/POS
P[2158]{
   GP1:
	UF : 7, UT : 3,	CONFIG : 'F U T, 0, 0, 0',
	X =   169.241  mm,	Y =   268.585  mm,	Z =     0.000  mm,
	W =  -167.363 deg,	P =     0.002 deg,	R =   163.143 deg
};
P[2159]{
   GP1:
	UF : 7, UT : 3,	CONFIG : 'F U T, 0, 0, 0',
	X =   183.720  mm,	Y =   258.920  mm,	Z =     0.001  mm,
	W =  -167.363 deg,	P =     0.001 deg,	R =   159.718 deg
};
P[2160]{
   GP1:
	UF : 7, UT : 3,	CONFIG : 'F U T, 0, 0, 0',
	X =   198.126  mm,	Y =   248.045  mm,	Z =     0.001  mm,
	W =  -167.364 deg,	P =     0.000 deg,	R =   156.405 deg
};
P[2161]{
   GP1:
	UF : 7, UT : 3,	CONFIG : 'F U T, 0, 0, 0',
	X =   212.090  mm,	Y =   236.233  mm,	Z =     0.001  mm,
	W =  -167.364 deg,	P =    -0.002 deg,	R =   153.153 deg
};
P[2162]{
   GP1:
	UF : 7, UT : 3,	CONFIG : 'F U T, 0, 0, 0',
	X =   224.191  mm,	Y =   224.763  mm,	Z =     0.000  mm,
	W =  -167.364 deg,	P =    -0.003 deg,	R =   149.479 deg
};
P[2163]{
   GP1:
	UF : 7, UT : 3,	CONFIG : 'F U T, 0, 0, 0',
	X =   224.191  mm,	Y =   224.763  mm,	Z =     0.000  mm,
	W =  -167.364 deg,	P =    -0.003 deg,	R =   149.479 deg
};
P[2164]{
   GP1:
	UF : 7, UT : 3,	CONFIG : 'F U T, 0, 0, 0',
	X =   224.191  mm,	Y =   224.763  mm,	Z =     0.000  mm,
	W =  -167.364 deg,	P =    -0.003 deg,	R =   149.479 deg
};
P[2165]{
   GP1:
	UF : 7, UT : 3,	CONFIG : 'F U T, 0, 0, 0',
	X =   224.191  mm,	Y =   224.763  mm,	Z =     0.000  mm,
	W =  -167.364 deg,	P =    -0.003 deg,	R =   149.479 deg
};
P[2166]{
   GP1:
	UF : 7, UT : 3,	CONFIG : 'F U T, 0, 0, 0',
	X =   269.018  mm,	Y =   168.557  mm,	Z =     0.000  mm,
	W =  -167.363 deg,	P =     0.003 deg,	R =   137.473 deg
};
P[2167]{
   GP1:
	UF : 7, UT : 3,	CONFIG : 'F U T, 0, 0, 0',
	X =   269.018  mm,	Y =   168.557  mm,	Z =     0.000  mm,
	W =  -167.363 deg,	P =     0.003 deg,	R =   137.473 deg
};
P[2168]{
   GP1:
	UF : 7, UT : 3,	CONFIG : 'F U T, 0, 0, 0',
	X =   269.018  mm,	Y =   168.557  mm,	Z =     0.000  mm,
	W =  -167.363 deg,	P =     0.003 deg,	R =   137.473 deg
};
P[2169]{
   GP1:
	UF : 7, UT : 3,	CONFIG : 'F U T, 0, 0, 0',
	X =   269.018  mm,	Y =   168.557  mm,	Z =     0.000  mm,
	W =  -167.363 deg,	P =     0.003 deg,	R =   137.473 deg
};
P[2170]{
   GP1:
	UF : 7, UT : 3,	CONFIG : 'F U T, 0, 0, 0',
	X =   277.589  mm,	Y =   154.047  mm,	Z =     0.001  mm,
	W =  -167.363 deg,	P =     0.001 deg,	R =   134.070 deg
};
P[2171]{
   GP1:
	UF : 7, UT : 3,	CONFIG : 'F U T, 0, 0, 0',
	X =   285.805  mm,	Y =   138.195  mm,	Z =     0.001  mm,
	W =  -167.364 deg,	P =     0.000 deg,	R =   130.902 deg
};
P[2172]{
   GP1:
	UF : 7, UT : 3,	CONFIG : 'F U T, 0, 0, 0',
	X =   292.963  mm,	Y =   122.300  mm,	Z =     0.001  mm,
	W =  -167.364 deg,	P =    -0.001 deg,	R =   127.666 deg
};
P[2173]{
   GP1:
	UF : 7, UT : 3,	CONFIG : 'F U T, 0, 0, 0',
	X =   299.514  mm,	Y =   105.233  mm,	Z =     0.000  mm,
	W =  -167.364 deg,	P =    -0.003 deg,	R =   124.545 deg
};
P[2174]{
   GP1:
	UF : 7, UT : 3,	CONFIG : 'F U T, 0, 0, 0',
	X =   299.514  mm,	Y =   105.233  mm,	Z =     0.000  mm,
	W =  -167.364 deg,	P =    -0.003 deg,	R =   124.545 deg
};
P[2175]{
   GP1:
	UF : 7, UT : 3,	CONFIG : 'F U T, 0, 0, 0',
	X =   299.514  mm,	Y =   105.233  mm,	Z =     0.000  mm,
	W =  -167.364 deg,	P =    -0.003 deg,	R =   124.545 deg
};
P[2176]{
   GP1:
	UF : 7, UT : 3,	CONFIG : 'F U T, 0, 0, 0',
	X =   299.514  mm,	Y =   105.233  mm,	Z =     0.000  mm,
	W =  -167.364 deg,	P =    -0.003 deg,	R =   124.545 deg
};
P[2177]{
   GP1:
	UF : 7, UT : 3,	CONFIG : 'F U T, 0, 0, 0',
	X =   315.526  mm,	Y =    35.143  mm,	Z =     0.000  mm,
	W =  -167.363 deg,	P =     0.001 deg,	R =   110.775 deg
};
P[2178]{
   GP1:
	UF : 7, UT : 3,	CONFIG : 'F U T, 0, 0, 0',
	X =   315.526  mm,	Y =    35.143  mm,	Z =     0.000  mm,
	W =  -167.363 deg,	P =     0.001 deg,	R =   110.775 deg
};
P[2179]{
   GP1:
	UF : 7, UT : 3,	CONFIG : 'F U T, 0, 0, 0',
	X =   315.526  mm,	Y =    35.143  mm,	Z =     0.000  mm,
	W =  -167.363 deg,	P =     0.001 deg,	R =   110.775 deg
};
P[2180]{
   GP1:
	UF : 7, UT : 3,	CONFIG : 'F U T, 0, 0, 0',
	X =   315.526  mm,	Y =    35.143  mm,	Z =     0.000  mm,
	W =  -167.363 deg,	P =     0.001 deg,	R =   110.775 deg
};
P[2181]{
   GP1:
	UF : 7, UT : 3,	CONFIG : 'F U T, 0, 0, 0',
	X =   316.958  mm,	Y =    17.828  mm,	Z =     0.000  mm,
	W =  -167.363 deg,	P =     0.000 deg,	R =   108.286 deg
};
P[2182]{
   GP1:
	UF : 7, UT : 3,	CONFIG : 'F U T, 0, 0, 0',
	X =   317.478  mm,	Y =     0.000  mm,	Z =     0.000  mm,
	W =  -167.364 deg,	P =    -0.001 deg,	R =   105.693 deg
};
P[2183]{
   GP1:
	UF : 7, UT : 3,	CONFIG : 'F U T, 0, 0, 0',
	X =   317.478  mm,	Y =     0.000  mm,	Z =     0.000  mm,
	W =  -167.364 deg,	P =    -0.001 deg,	R =   105.693 deg
};
P[2184]{
   GP1:
	UF : 7, UT : 3,	CONFIG : 'F U T, 0, 0, 0',
	X =   317.478  mm,	Y =     0.000  mm,	Z =     0.000  mm,
	W =  -167.364 deg,	P =    -0.001 deg,	R =   105.693 deg
};
P[2185]{
   GP1:
	UF : 7, UT : 3,	CONFIG : 'F U T, 0, 0, 0',
	X =   317.478  mm,	Y =     0.000  mm,	Z =     0.000  mm,
	W =  -167.364 deg,	P =    -0.001 deg,	R =   105.693 deg
};
P[2186]{
   GP1:
	UF : 7, UT : 3,	CONFIG : 'F U T, 0, 0, 0',
	X =   314.344  mm,	Y =     0.000  mm,	Z =     0.000  mm,
	W =  -167.364 deg,	P =    -0.001 deg,	R =   105.705 deg
};
P[2187]{
   GP1:
	UF : 7, UT : 3,	CONFIG : 'F U T, 0, 0, 0',
	X =   314.344  mm,	Y =     0.000  mm,	Z =     0.000  mm,
	W =  -167.364 deg,	P =    -0.001 deg,	R =   105.705 deg
};
P[2188]{
   GP1:
	UF : 7, UT : 3,	CONFIG : 'F U T, 0, 0, 0',
	X =   314.344  mm,	Y =     0.000  mm,	Z =     0.000  mm,
	W =  -167.364 deg,	P =    -0.001 deg,	R =   105.705 deg
};
P[2189]{
   GP1:
	UF : 7, UT : 3,	CONFIG : 'F U T, 0, 0, 0',
	X =   314.344  mm,	Y =     0.000  mm,	Z =     0.000  mm,
	W =  -167.364 deg,	P =    -0.001 deg,	R =   105.705 deg
};
P[2190]{
   GP1:
	UF : 7, UT : 3,	CONFIG : 'F U T, 0, 0, 0',
	X =   313.796  mm,	Y =    18.258  mm,	Z =     0.000  mm,
	W =  -167.363 deg,	P =     0.000 deg,	R =   108.359 deg
};
P[2191]{
   GP1:
	UF : 7, UT : 3,	CONFIG : 'F U T, 0, 0, 0',
	X =   312.363  mm,	Y =    35.193  mm,	Z =     0.000  mm,
	W =  -167.363 deg,	P =     0.001 deg,	R =   111.081 deg
};
P[2192]{
   GP1:
	UF : 7, UT : 3,	CONFIG : 'F U T, 0, 0, 0',
	X =   312.363  mm,	Y =    35.193  mm,	Z =     0.000  mm,
	W =  -167.363 deg,	P =     0.001 deg,	R =   111.081 deg
};
P[2193]{
   GP1:
	UF : 7, UT : 3,	CONFIG : 'F U T, 0, 0, 0',
	X =   312.363  mm,	Y =    35.193  mm,	Z =     0.000  mm,
	W =  -167.363 deg,	P =     0.001 deg,	R =   111.081 deg
};
P[2194]{
   GP1:
	UF : 7, UT : 3,	CONFIG : 'F U T, 0, 0, 0',
	X =   312.363  mm,	Y =    35.193  mm,	Z =     0.000  mm,
	W =  -167.363 deg,	P =     0.001 deg,	R =   111.081 deg
};
P[2195]{
   GP1:
	UF : 7, UT : 3,	CONFIG : 'F U T, 0, 0, 0',
	X =   296.692  mm,	Y =   103.818  mm,	Z =     0.000  mm,
	W =  -167.364 deg,	P =    -0.003 deg,	R =   124.612 deg
};
P[2196]{
   GP1:
	UF : 7, UT : 3,	CONFIG : 'F U T, 0, 0, 0',
	X =   296.692  mm,	Y =   103.818  mm,	Z =     0.000  mm,
	W =  -167.364 deg,	P =    -0.003 deg,	R =   124.612 deg
};
P[2197]{
   GP1:
	UF : 7, UT : 3,	CONFIG : 'F U T, 0, 0, 0',
	X =   296.692  mm,	Y =   103.818  mm,	Z =     0.000  mm,
	W =  -167.364 deg,	P =    -0.003 deg,	R =   124.612 deg
};
P[2198]{
   GP1:
	UF : 7, UT : 3,	CONFIG : 'F U T, 0, 0, 0',
	X =   296.692  mm,	Y =   103.818  mm,	Z =     0.000  mm,
	W =  -167.364 deg,	P =    -0.003 deg,	R =   124.612 deg
};
P[2199]{
   GP1:
	UF : 7, UT : 3,	CONFIG : 'F U T, 0, 0, 0',
	X =   289.976  mm,	Y =   121.319  mm,	Z =     0.001  mm,
	W =  -167.364 deg,	P =    -0.001 deg,	R =   127.739 deg
};
P[2200]{
   GP1:
	UF : 7, UT : 3,	CONFIG : 'F U T, 0, 0, 0',
	X =   282.724  mm,	Y =   137.365  mm,	Z =     0.001  mm,
	W =  -167.363 deg,	P =     0.000 deg,	R =   130.985 deg
};
P[2201]{
   GP1:
	UF : 7, UT : 3,	CONFIG : 'F U T, 0, 0, 0',
	X =   274.534  mm,	Y =   153.088  mm,	Z =     0.001  mm,
	W =  -167.363 deg,	P =     0.001 deg,	R =   134.198 deg
};
P[2202]{
   GP1:
	UF : 7, UT : 3,	CONFIG : 'F U T, 0, 0, 0',
	X =   266.148  mm,	Y =   167.232  mm,	Z =     0.000  mm,
	W =  -167.362 deg,	P =     0.003 deg,	R =   137.749 deg
};
P[2203]{
   GP1:
	UF : 7, UT : 3,	CONFIG : 'F U T, 0, 0, 0',
	X =   266.148  mm,	Y =   167.232  mm,	Z =     0.000  mm,
	W =  -167.362 deg,	P =     0.003 deg,	R =   137.749 deg
};
P[2204]{
   GP1:
	UF : 7, UT : 3,	CONFIG : 'F U T, 0, 0, 0',
	X =   266.148  mm,	Y =   167.232  mm,	Z =     0.000  mm,
	W =  -167.362 deg,	P =     0.003 deg,	R =   137.749 deg
};
P[2205]{
   GP1:
	UF : 7, UT : 3,	CONFIG : 'F U T, 0, 0, 0',
	X =   266.148  mm,	Y =   167.232  mm,	Z =     0.000  mm,
	W =  -167.362 deg,	P =     0.003 deg,	R =   137.749 deg
};
P[2206]{
   GP1:
	UF : 7, UT : 3,	CONFIG : 'F U T, 0, 0, 0',
	X =   222.261  mm,	Y =   222.261  mm,	Z =     0.000  mm,
	W =  -167.364 deg,	P =    -0.003 deg,	R =   149.599 deg
};
P[2207]{
   GP1:
	UF : 7, UT : 3,	CONFIG : 'F U T, 0, 0, 0',
	X =   222.261  mm,	Y =   222.261  mm,	Z =     0.000  mm,
	W =  -167.364 deg,	P =    -0.003 deg,	R =   149.599 deg
};
P[2208]{
   GP1:
	UF : 7, UT : 3,	CONFIG : 'F U T, 0, 0, 0',
	X =   222.261  mm,	Y =   222.261  mm,	Z =     0.000  mm,
	W =  -167.364 deg,	P =    -0.003 deg,	R =   149.599 deg
};
P[2209]{
   GP1:
	UF : 7, UT : 3,	CONFIG : 'F U T, 0, 0, 0',
	X =   222.261  mm,	Y =   222.261  mm,	Z =     0.000  mm,
	W =  -167.364 deg,	P =    -0.003 deg,	R =   149.599 deg
};
P[2210]{
   GP1:
	UF : 7, UT : 3,	CONFIG : 'F U T, 0, 0, 0',
	X =   209.897  mm,	Y =   233.994  mm,	Z =     0.001  mm,
	W =  -167.364 deg,	P =    -0.002 deg,	R =   153.153 deg
};
P[2211]{
   GP1:
	UF : 7, UT : 3,	CONFIG : 'F U T, 0, 0, 0',
	X =   195.899  mm,	Y =   245.814  mm,	Z =     0.001  mm,
	W =  -167.363 deg,	P =     0.000 deg,	R =   156.411 deg
};
P[2212]{
   GP1:
	UF : 7, UT : 3,	CONFIG : 'F U T, 0, 0, 0',
	X =   181.688  mm,	Y =   256.510  mm,	Z =     0.001  mm,
	W =  -167.363 deg,	P =     0.001 deg,	R =   159.771 deg
};
P[2213]{
   GP1:
	UF : 7, UT : 3,	CONFIG : 'F U T, 0, 0, 0',
	X =   167.232  mm,	Y =   266.148  mm,	Z =     0.000  mm,
	W =  -167.362 deg,	P =     0.002 deg,	R =   163.242 deg
};
P[2214]{
   GP1:
	UF : 7, UT : 3,	CONFIG : 'F U T, 0, 0, 0',
	X =   167.232  mm,	Y =   266.148  mm,	Z =     0.000  mm,
	W =  -167.362 deg,	P =     0.002 deg,	R =   163.242 deg
};
P[2215]{
   GP1:
	UF : 7, UT : 3,	CONFIG : 'F U T, 0, 0, 0',
	X =   167.232  mm,	Y =   266.148  mm,	Z =     0.000  mm,
	W =  -167.362 deg,	P =     0.002 deg,	R =   163.242 deg
};
P[2216]{
   GP1:
	UF : 7, UT : 3,	CONFIG : 'F U T, 0, 0, 0',
	X =   167.232  mm,	Y =   266.148  mm,	Z =     0.000  mm,
	W =  -167.362 deg,	P =     0.002 deg,	R =   163.242 deg
};
P[2217]{
   GP1:
	UF : 7, UT : 3,	CONFIG : 'F U T, 0, 0, 0',
	X =   103.816  mm,	Y =   296.692  mm,	Z =     0.000  mm,
	W =  -167.364 deg,	P =    -0.001 deg,	R =   175.609 deg
};
P[2218]{
   GP1:
	UF : 7, UT : 3,	CONFIG : 'F U T, 0, 0, 0',
	X =   103.816  mm,	Y =   296.692  mm,	Z =     0.000  mm,
	W =  -167.364 deg,	P =    -0.001 deg,	R =   175.609 deg
};
P[2219]{
   GP1:
	UF : 7, UT : 3,	CONFIG : 'F U T, 0, 0, 0',
	X =   103.816  mm,	Y =   296.692  mm,	Z =     0.000  mm,
	W =  -167.364 deg,	P =    -0.001 deg,	R =   175.609 deg
};
P[2220]{
   GP1:
	UF : 7, UT : 3,	CONFIG : 'F U T, 0, 0, 0',
	X =   103.816  mm,	Y =   296.692  mm,	Z =     0.000  mm,
	W =  -167.364 deg,	P =    -0.001 deg,	R =   175.609 deg
};
P[2221]{
   GP1:
	UF : 7, UT : 3,	CONFIG : 'F U T, 0, 0, 0',
	X =    87.953  mm,	Y =   301.775  mm,	Z =     0.000  mm,
	W =  -167.364 deg,	P =    -0.001 deg,	R =   178.852 deg
};
P[2222]{
   GP1:
	UF : 7, UT : 3,	CONFIG : 'F U T, 0, 0, 0',
	X =    71.164  mm,	Y =   306.169  mm,	Z =     0.000  mm,
	W =  -167.363 deg,	P =     0.000 deg,	R =  -178.042 deg
};
P[2223]{
   GP1:
	UF : 7, UT : 3,	CONFIG : 'F U T, 0, 0, 0',
	X =    54.389  mm,	Y =   309.594  mm,	Z =     0.000  mm,
	W =  -167.363 deg,	P =     0.000 deg,	R =  -174.890 deg
};
P[2224]{
   GP1:
	UF : 7, UT : 3,	CONFIG : 'F U T, 0, 0, 0',
	X =    35.197  mm,	Y =   312.362  mm,	Z =     0.000  mm,
	W =  -167.363 deg,	P =     0.001 deg,	R =  -171.894 deg
};
P[2225]{
   GP1:
	UF : 7, UT : 3,	CONFIG : 'F U T, 0, 0, 0',
	X =    35.197  mm,	Y =   312.362  mm,	Z =     0.000  mm,
	W =  -167.363 deg,	P =     0.001 deg,	R =  -171.894 deg
};
P[2226]{
   GP1:
	UF : 7, UT : 3,	CONFIG : 'F U T, 0, 0, 0',
	X =    35.197  mm,	Y =   312.362  mm,	Z =     0.000  mm,
	W =  -167.363 deg,	P =     0.001 deg,	R =  -171.894 deg
};
P[2227]{
   GP1:
	UF : 7, UT : 3,	CONFIG : 'F U T, 0, 0, 0',
	X =    35.197  mm,	Y =   312.362  mm,	Z =     0.000  mm,
	W =  -167.363 deg,	P =     0.001 deg,	R =  -171.894 deg
};
P[2228]{
   GP1:
	UF : 7, UT : 3,	CONFIG : 'F U T, 0, 0, 0',
	X =   -35.197  mm,	Y =   312.362  mm,	Z =     0.000  mm,
	W =  -167.364 deg,	P =    -0.001 deg,	R =  -157.993 deg
};
P[2229]{
   GP1:
	UF : 7, UT : 3,	CONFIG : 'F U T, 0, 0, 0',
	X =   -35.197  mm,	Y =   312.362  mm,	Z =     0.000  mm,
	W =  -167.364 deg,	P =    -0.001 deg,	R =  -157.993 deg
};
P[2230]{
   GP1:
	UF : 7, UT : 3,	CONFIG : 'F U T, 0, 0, 0',
	X =   -35.197  mm,	Y =   312.362  mm,	Z =     0.000  mm,
	W =  -167.364 deg,	P =    -0.001 deg,	R =  -157.993 deg
};
P[2231]{
   GP1:
	UF : 7, UT : 3,	CONFIG : 'F U T, 0, 0, 0',
	X =   -35.197  mm,	Y =   312.362  mm,	Z =     0.000  mm,
	W =  -167.364 deg,	P =    -0.001 deg,	R =  -157.993 deg
};
P[2232]{
   GP1:
	UF : 7, UT : 3,	CONFIG : 'F U T, 0, 0, 0',
	X =   -54.397  mm,	Y =   309.592  mm,	Z =     0.001  mm,
	W =  -167.363 deg,	P =     0.000 deg,	R =  -154.999 deg
};
P[2233]{
   GP1:
	UF : 7, UT : 3,	CONFIG : 'F U T, 0, 0, 0',
	X =   -71.123  mm,	Y =   306.179  mm,	Z =     0.001  mm,
	W =  -167.363 deg,	P =     0.002 deg,	R =  -151.872 deg
};
P[2234]{
   GP1:
	UF : 7, UT : 3,	CONFIG : 'F U T, 0, 0, 0',
	X =   -87.830  mm,	Y =   301.810  mm,	Z =     0.001  mm,
	W =  -167.362 deg,	P =     0.003 deg,	R =  -148.771 deg
};
P[2235]{
   GP1:
	UF : 7, UT : 3,	CONFIG : 'F U T, 0, 0, 0',
	X =  -103.816  mm,	Y =   296.692  mm,	Z =     0.000  mm,
	W =  -167.361 deg,	P =     0.004 deg,	R =  -145.598 deg
};
P[2236]{
   GP1:
	UF : 7, UT : 3,	CONFIG : 'F U T, 0, 0, 0',
	X =  -103.816  mm,	Y =   296.692  mm,	Z =     0.000  mm,
	W =  -167.361 deg,	P =     0.004 deg,	R =  -145.598 deg
};
P[2237]{
   GP1:
	UF : 7, UT : 3,	CONFIG : 'F U T, 0, 0, 0',
	X =  -103.816  mm,	Y =   296.692  mm,	Z =     0.000  mm,
	W =  -167.361 deg,	P =     0.004 deg,	R =  -145.598 deg
};
P[2238]{
   GP1:
	UF : 7, UT : 3,	CONFIG : 'F U T, 0, 0, 0',
	X =  -103.816  mm,	Y =   296.692  mm,	Z =     0.000  mm,
	W =  -167.361 deg,	P =     0.004 deg,	R =  -145.598 deg
};
P[2239]{
   GP1:
	UF : 7, UT : 3,	CONFIG : 'F U T, 0, 0, 0',
	X =  -167.232  mm,	Y =   266.148  mm,	Z =     0.000  mm,
	W =  -167.365 deg,	P =    -0.022 deg,	R =  -132.938 deg
};
P[2240]{
   GP1:
	UF : 7, UT : 3,	CONFIG : 'F U T, 0, 0, 0',
	X =  -167.232  mm,	Y =   266.148  mm,	Z =     0.000  mm,
	W =  -167.365 deg,	P =    -0.022 deg,	R =  -132.938 deg
};
P[2241]{
   GP1:
	UF : 7, UT : 3,	CONFIG : 'F U T, 0, 0, 0',
	X =  -167.232  mm,	Y =   266.148  mm,	Z =     0.000  mm,
	W =  -167.365 deg,	P =    -0.022 deg,	R =  -132.938 deg
};
P[2242]{
   GP1:
	UF : 7, UT : 3,	CONFIG : 'F U T, 0, 0, 0',
	X =  -167.232  mm,	Y =   266.148  mm,	Z =     0.000  mm,
	W =  -167.365 deg,	P =    -0.022 deg,	R =  -132.938 deg
};
P[2243]{
   GP1:
	UF : 7, UT : 3,	CONFIG : 'F U T, 0, 0, 0',
	X =  -183.114  mm,	Y =   255.488  mm,	Z =     0.011  mm,
	W =  -167.354 deg,	P =    -0.024 deg,	R =  -129.291 deg
};
P[2244]{
   GP1:
	UF : 7, UT : 3,	CONFIG : 'F U T, 0, 0, 0',
	X =  -198.763  mm,	Y =   243.515  mm,	Z =     0.023  mm,
	W =  -167.343 deg,	P =    -0.029 deg,	R =  -125.737 deg
};
P[2245]{
   GP1:
	UF : 7, UT : 3,	CONFIG : 'F U T, 0, 0, 0',
	X =  -211.069  mm,	Y =   232.923  mm,	Z =     0.022  mm,
	W =  -167.329 deg,	P =     0.048 deg,	R =  -122.698 deg
};
P[2246]{
   GP1:
	UF : 7, UT : 3,	CONFIG : 'F U T, 0, 0, 0',
	X =  -222.261  mm,	Y =   222.261  mm,	Z =     0.000  mm,
	W =  -167.307 deg,	P =     0.119 deg,	R =  -119.437 deg
};
P[2247]{
   GP1:
	UF : 7, UT : 3,	CONFIG : 'F U T, 0, 0, 0',
	X =  -222.261  mm,	Y =   222.261  mm,	Z =     0.000  mm,
	W =  -167.307 deg,	P =     0.119 deg,	R =  -119.437 deg
};
P[2248]{
   GP1:
	UF : 7, UT : 3,	CONFIG : 'F U T, 0, 0, 0',
	X =  -222.261  mm,	Y =   222.261  mm,	Z =     0.000  mm,
	W =  -167.307 deg,	P =     0.119 deg,	R =  -119.437 deg
};
P[2249]{
   GP1:
	UF : 7, UT : 3,	CONFIG : 'F U T, 0, 0, 0',
	X =  -222.261  mm,	Y =   222.261  mm,	Z =     0.000  mm,
	W =  -167.307 deg,	P =     0.119 deg,	R =  -119.437 deg
};
P[2250]{
   GP1:
	UF : 7, UT : 3,	CONFIG : 'F U T, 0, 0, 0',
	X =  -266.148  mm,	Y =   167.232  mm,	Z =     0.000  mm,
	W =  -167.451 deg,	P =    -1.057 deg,	R =  -107.603 deg
};
P[2251]{
   GP1:
	UF : 7, UT : 3,	CONFIG : 'F U T, 0, 0, 0',
	X =  -266.148  mm,	Y =   167.232  mm,	Z =     0.000  mm,
	W =  -167.451 deg,	P =    -1.057 deg,	R =  -107.603 deg
};
P[2252]{
   GP1:
	UF : 7, UT : 3,	CONFIG : 'F U T, 0, 0, 0',
	X =  -266.148  mm,	Y =   167.232  mm,	Z =     0.000  mm,
	W =  -167.451 deg,	P =    -1.057 deg,	R =  -107.603 deg
};
P[2253]{
   GP1:
	UF : 7, UT : 3,	CONFIG : 'F U T, 0, 0, 0',
	X =  -266.148  mm,	Y =   167.232  mm,	Z =     0.000  mm,
	W =  -167.451 deg,	P =    -1.057 deg,	R =  -107.603 deg
};
P[2254]{
   GP1:
	UF : 7, UT : 3,	CONFIG : 'F U T, 0, 0, 0',
	X =  -269.323  mm,	Y =   162.065  mm,	Z =     0.117  mm,
	W =  -167.681 deg,	P =    -1.097 deg,	R =  -105.987 deg
};
P[2255]{
   GP1:
	UF : 7, UT : 3,	CONFIG : 'F U T, 0, 0, 0',
	X =  -277.022  mm,	Y =   148.536  mm,	Z =     0.388  mm,
	W =  -168.155 deg,	P =    -0.523 deg,	R =  -103.206 deg
};
P[2256]{
   GP1:
	UF : 7, UT : 3,	CONFIG : 'F U T, 0, 0, 0',
	X =  -285.722  mm,	Y =   131.011  mm,	Z =     0.439  mm,
	W =  -168.148 deg,	P =     0.621 deg,	R =   -99.624 deg
};
P[2257]{
   GP1:
	UF : 7, UT : 3,	CONFIG : 'F U T, 0, 0, 0',
	X =  -290.703  mm,	Y =   119.560  mm,	Z =     0.270  mm,
	W =  -167.700 deg,	P =     1.177 deg,	R =   -97.280 deg
};
P[2258]{
   GP1:
	UF : 7, UT : 3,	CONFIG : 'F U T, 0, 0, 0',
	X =  -292.713  mm,	Y =   114.575  mm,	Z =     0.169  mm,
	W =  -167.445 deg,	P =     1.139 deg,	R =   -96.303 deg
};
P[2259]{
   GP1:
	UF : 7, UT : 3,	CONFIG : 'F U T, 0, 0, 0',
	X =  -296.692  mm,	Y =   103.818  mm,	Z =     0.000  mm,
	W =  -167.160 deg,	P =     0.453 deg,	R =   -94.516 deg
};
P[2260]{
   GP1:
	UF : 7, UT : 3,	CONFIG : 'F U T, 0, 0, 0',
	X =  -296.692  mm,	Y =   103.818  mm,	Z =     0.000  mm,
	W =  -167.160 deg,	P =     0.453 deg,	R =   -94.516 deg
};
P[2261]{
   GP1:
	UF : 7, UT : 3,	CONFIG : 'F U T, 0, 0, 0',
	X =  -296.692  mm,	Y =   103.818  mm,	Z =     0.000  mm,
	W =  -167.160 deg,	P =     0.453 deg,	R =   -94.516 deg
};
P[2262]{
   GP1:
	UF : 7, UT : 3,	CONFIG : 'F U T, 0, 0, 0',
	X =  -296.692  mm,	Y =   103.818  mm,	Z =     0.000  mm,
	W =  -167.160 deg,	P =     0.453 deg,	R =   -94.516 deg
};
P[2263]{
   GP1:
	UF : 7, UT : 3,	CONFIG : 'F U T, 0, 1, 0',
	X =  -312.363  mm,	Y =    35.193  mm,	Z =     0.000  mm,
	W =  -167.364 deg,	P =    -0.010 deg,	R =   -80.974 deg
};
P[2264]{
   GP1:
	UF : 7, UT : 3,	CONFIG : 'F U T, 0, 1, 0',
	X =  -312.363  mm,	Y =    35.193  mm,	Z =     0.000  mm,
	W =  -167.364 deg,	P =    -0.010 deg,	R =   -80.974 deg
};
P[2265]{
   GP1:
	UF : 7, UT : 3,	CONFIG : 'F U T, 0, 1, 0',
	X =  -312.363  mm,	Y =    35.193  mm,	Z =     0.000  mm,
	W =  -167.364 deg,	P =    -0.010 deg,	R =   -80.974 deg
};
P[2266]{
   GP1:
	UF : 7, UT : 3,	CONFIG : 'F U T, 0, 1, 0',
	X =  -312.363  mm,	Y =    35.193  mm,	Z =     0.000  mm,
	W =  -167.364 deg,	P =    -0.010 deg,	R =   -80.974 deg
};
P[2267]{
   GP1:
	UF : 7, UT : 3,	CONFIG : 'F U T, 0, 1, 0',
	X =  -313.784  mm,	Y =    18.505  mm,	Z =     0.001  mm,
	W =  -167.364 deg,	P =    -0.002 deg,	R =   -78.279 deg
};
P[2268]{
   GP1:
	UF : 7, UT : 3,	CONFIG : 'F U T, 0, 1, 0',
	X =  -314.344  mm,	Y =     0.000  mm,	Z =     0.000  mm,
	W =  -167.362 deg,	P =     0.006 deg,	R =   -75.585 deg
};
P[2269]{
   GP1:
	UF : 7, UT : 3,	CONFIG : 'F U T, 0, 1, 0',
	X =  -314.344  mm,	Y =     0.000  mm,	Z =     0.000  mm,
	W =  -167.362 deg,	P =     0.006 deg,	R =   -75.585 deg
};
P[2270]{
   GP1:
	UF : 7, UT : 3,	CONFIG : 'F U T, 0, 1, 0',
	X =  -314.344  mm,	Y =     0.000  mm,	Z =     0.000  mm,
	W =  -167.362 deg,	P =     0.006 deg,	R =   -75.585 deg
};
P[2271]{
   GP1:
	UF : 7, UT : 3,	CONFIG : 'F U T, 0, 1, 0',
	X =  -314.344  mm,	Y =     0.000  mm,	Z =     0.000  mm,
	W =  -167.362 deg,	P =     0.006 deg,	R =   -75.585 deg
};
P[2272]{
   GP1:
	UF : 7, UT : 3,	CONFIG : 'F U T, 0, 1, 0',
	X =  -311.210  mm,	Y =     0.000  mm,	Z =     0.000  mm,
	W =  -167.362 deg,	P =     0.005 deg,	R =   -75.574 deg
};
P[2273]{
   GP1:
	UF : 7, UT : 3,	CONFIG : 'F U T, 0, 1, 0',
	X =  -311.210  mm,	Y =     0.000  mm,	Z =     0.000  mm,
	W =  -167.362 deg,	P =     0.005 deg,	R =   -75.574 deg
};
P[2274]{
   GP1:
	UF : 7, UT : 3,	CONFIG : 'F U T, 0, 1, 0',
	X =  -311.210  mm,	Y =     0.000  mm,	Z =     0.000  mm,
	W =  -167.362 deg,	P =     0.005 deg,	R =   -75.574 deg
};
P[2275]{
   GP1:
	UF : 7, UT : 3,	CONFIG : 'F U T, 0, 1, 0',
	X =  -311.210  mm,	Y =     0.000  mm,	Z =     0.000  mm,
	W =  -167.362 deg,	P =     0.005 deg,	R =   -75.574 deg
};
P[2276]{
   GP1:
	UF : 7, UT : 3,	CONFIG : 'F U T, 0, 1, 0',
	X =  -310.609  mm,	Y =    19.167  mm,	Z =     0.001  mm,
	W =  -167.363 deg,	P =    -0.003 deg,	R =   -78.435 deg
};
P[2277]{
   GP1:
	UF : 7, UT : 3,	CONFIG : 'F U T, 0, 1, 0',
	X =  -309.165  mm,	Y =    35.521  mm,	Z =     0.000  mm,
	W =  -167.364 deg,	P =    -0.010 deg,	R =   -81.404 deg
};
P[2278]{
   GP1:
	UF : 7, UT : 3,	CONFIG : 'F U T, 0, 1, 0',
	X =  -309.165  mm,	Y =    35.521  mm,	Z =     0.000  mm,
	W =  -167.364 deg,	P =    -0.010 deg,	R =   -81.404 deg
};
P[2279]{
   GP1:
	UF : 7, UT : 3,	CONFIG : 'F U T, 0, 1, 0',
	X =  -309.165  mm,	Y =    35.521  mm,	Z =     0.000  mm,
	W =  -167.364 deg,	P =    -0.010 deg,	R =   -81.404 deg
};
P[2280]{
   GP1:
	UF : 7, UT : 3,	CONFIG : 'F U T, 0, 1, 0',
	X =  -309.165  mm,	Y =    35.521  mm,	Z =     0.000  mm,
	W =  -167.364 deg,	P =    -0.010 deg,	R =   -81.404 deg
};
P[2281]{
   GP1:
	UF : 7, UT : 3,	CONFIG : 'F U T, 0, 0, 0',
	X =  -293.963  mm,	Y =   102.140  mm,	Z =     0.000  mm,
	W =  -167.168 deg,	P =     0.349 deg,	R =   -94.592 deg
};
P[2282]{
   GP1:
	UF : 7, UT : 3,	CONFIG : 'F U T, 0, 0, 0',
	X =  -293.963  mm,	Y =   102.140  mm,	Z =     0.000  mm,
	W =  -167.168 deg,	P =     0.349 deg,	R =   -94.592 deg
};
P[2283]{
   GP1:
	UF : 7, UT : 3,	CONFIG : 'F U T, 0, 0, 0',
	X =  -293.963  mm,	Y =   102.140  mm,	Z =     0.000  mm,
	W =  -167.168 deg,	P =     0.349 deg,	R =   -94.592 deg
};
P[2284]{
   GP1:
	UF : 7, UT : 3,	CONFIG : 'F U T, 0, 0, 0',
	X =  -293.963  mm,	Y =   102.140  mm,	Z =     0.000  mm,
	W =  -167.168 deg,	P =     0.349 deg,	R =   -94.592 deg
};
P[2285]{
   GP1:
	UF : 7, UT : 3,	CONFIG : 'F U T, 0, 0, 0',
	X =  -289.713  mm,	Y =   113.629  mm,	Z =     0.153  mm,
	W =  -167.448 deg,	P =     0.997 deg,	R =   -96.337 deg
};
P[2286]{
   GP1:
	UF : 7, UT : 3,	CONFIG : 'F U T, 0, 0, 0',
	X =  -285.444  mm,	Y =   123.944  mm,	Z =     0.328  mm,
	W =  -167.908 deg,	P =     0.905 deg,	R =   -98.395 deg
};
P[2287]{
   GP1:
	UF : 7, UT : 3,	CONFIG : 'F U T, 0, 0, 0',
	X =  -278.233  mm,	Y =   139.399  mm,	Z =     0.413  mm,
	W =  -168.175 deg,	P =     0.054 deg,	R =  -101.560 deg
};
P[2288]{
   GP1:
	UF : 7, UT : 3,	CONFIG : 'F U T, 0, 0, 0',
	X =  -270.057  mm,	Y =   154.632  mm,	Z =     0.235  mm,
	W =  -167.853 deg,	P =    -0.831 deg,	R =  -104.757 deg
};
P[2289]{
   GP1:
	UF : 7, UT : 3,	CONFIG : 'F U T, 0, 0, 0',
	X =  -263.128  mm,	Y =   166.143  mm,	Z =     0.000  mm,
	W =  -167.353 deg,	P =    -0.982 deg,	R =  -107.921 deg
};
P[2290]{
   GP1:
	UF : 7, UT : 3,	CONFIG : 'F U T, 0, 0, 0',
	X =  -263.128  mm,	Y =   166.143  mm,	Z =     0.000  mm,
	W =  -167.353 deg,	P =    -0.982 deg,	R =  -107.921 deg
};
P[2291]{
   GP1:
	UF : 7, UT : 3,	CONFIG : 'F U T, 0, 0, 0',
	X =  -263.128  mm,	Y =   166.143  mm,	Z =     0.000  mm,
	W =  -167.353 deg,	P =    -0.982 deg,	R =  -107.921 deg
};
P[2292]{
   GP1:
	UF : 7, UT : 3,	CONFIG : 'F U T, 0, 0, 0',
	X =  -263.128  mm,	Y =   166.143  mm,	Z =     0.000  mm,
	W =  -167.353 deg,	P =    -0.982 deg,	R =  -107.921 deg
};
P[2293]{
   GP1:
	UF : 7, UT : 3,	CONFIG : 'F U T, 0, 0, 0',
	X =  -220.529  mm,	Y =   219.561  mm,	Z =     0.000  mm,
	W =  -167.294 deg,	P =     0.118 deg,	R =  -119.493 deg
};
P[2294]{
   GP1:
	UF : 7, UT : 3,	CONFIG : 'F U T, 0, 0, 0',
	X =  -220.529  mm,	Y =   219.561  mm,	Z =     0.000  mm,
	W =  -167.294 deg,	P =     0.118 deg,	R =  -119.493 deg
};
P[2295]{
   GP1:
	UF : 7, UT : 3,	CONFIG : 'F U T, 0, 0, 0',
	X =  -220.529  mm,	Y =   219.561  mm,	Z =     0.000  mm,
	W =  -167.294 deg,	P =     0.118 deg,	R =  -119.493 deg
};
P[2296]{
   GP1:
	UF : 7, UT : 3,	CONFIG : 'F U T, 0, 0, 0',
	X =  -220.529  mm,	Y =   219.561  mm,	Z =     0.000  mm,
	W =  -167.294 deg,	P =     0.118 deg,	R =  -119.493 deg
};
P[2297]{
   GP1:
	UF : 7, UT : 3,	CONFIG : 'F U T, 0, 0, 0',
	X =  -208.972  mm,	Y =   230.595  mm,	Z =     0.023  mm,
	W =  -167.322 deg,	P =     0.047 deg,	R =  -122.742 deg
};
P[2298]{
   GP1:
	UF : 7, UT : 3,	CONFIG : 'F U T, 0, 0, 0',
	X =  -196.378  mm,	Y =   241.419  mm,	Z =     0.024  mm,
	W =  -167.342 deg,	P =    -0.031 deg,	R =  -125.847 deg
};
P[2299]{
   GP1:
	UF : 7, UT : 3,	CONFIG : 'F U T, 0, 0, 0',
	X =  -181.152  mm,	Y =   253.038  mm,	Z =     0.012  mm,
	W =  -167.352 deg,	P =    -0.027 deg,	R =  -129.328 deg
};
P[2300]{
   GP1:
	UF : 7, UT : 3,	CONFIG : 'F U T, 0, 0, 0',
	X =  -164.987  mm,	Y =   263.859  mm,	Z =     0.000  mm,
	W =  -167.364 deg,	P =    -0.024 deg,	R =  -132.775 deg
};
P[2301]{
   GP1:
	UF : 7, UT : 3,	CONFIG : 'F U T, 0, 0, 0',
	X =  -164.987  mm,	Y =   263.859  mm,	Z =     0.000  mm,
	W =  -167.364 deg,	P =    -0.024 deg,	R =  -132.775 deg
};
P[2302]{
   GP1:
	UF : 7, UT : 3,	CONFIG : 'F U T, 0, 0, 0',
	X =  -164.987  mm,	Y =   263.859  mm,	Z =     0.000  mm,
	W =  -167.364 deg,	P =    -0.024 deg,	R =  -132.775 deg
};
P[2303]{
   GP1:
	UF : 7, UT : 3,	CONFIG : 'F U T, 0, 0, 0',
	X =  -164.987  mm,	Y =   263.859  mm,	Z =     0.000  mm,
	W =  -167.364 deg,	P =    -0.024 deg,	R =  -132.775 deg
};
P[2304]{
   GP1:
	UF : 7, UT : 3,	CONFIG : 'F U T, 0, 0, 0',
	X =  -103.426  mm,	Y =   293.504  mm,	Z =     0.000  mm,
	W =  -167.361 deg,	P =     0.005 deg,	R =  -145.207 deg
};
P[2305]{
   GP1:
	UF : 7, UT : 3,	CONFIG : 'F U T, 0, 0, 0',
	X =  -103.426  mm,	Y =   293.504  mm,	Z =     0.000  mm,
	W =  -167.361 deg,	P =     0.005 deg,	R =  -145.207 deg
};
P[2306]{
   GP1:
	UF : 7, UT : 3,	CONFIG : 'F U T, 0, 0, 0',
	X =  -103.426  mm,	Y =   293.504  mm,	Z =     0.000  mm,
	W =  -167.361 deg,	P =     0.005 deg,	R =  -145.207 deg
};
P[2307]{
   GP1:
	UF : 7, UT : 3,	CONFIG : 'F U T, 0, 0, 0',
	X =  -103.426  mm,	Y =   293.504  mm,	Z =     0.000  mm,
	W =  -167.361 deg,	P =     0.005 deg,	R =  -145.207 deg
};
P[2308]{
   GP1:
	UF : 7, UT : 3,	CONFIG : 'F U T, 0, 0, 0',
	X =   -87.653  mm,	Y =   298.599  mm,	Z =     0.001  mm,
	W =  -167.362 deg,	P =     0.003 deg,	R =  -148.621 deg
};
P[2309]{
   GP1:
	UF : 7, UT : 3,	CONFIG : 'F U T, 0, 0, 0',
	X =   -70.707  mm,	Y =   303.056  mm,	Z =     0.001  mm,
	W =  -167.362 deg,	P =     0.002 deg,	R =  -151.841 deg
};
P[2310]{
   GP1:
	UF : 7, UT : 3,	CONFIG : 'F U T, 0, 0, 0',
	X =   -53.533  mm,	Y =   306.560  mm,	Z =     0.001  mm,
	W =  -167.363 deg,	P =     0.000 deg,	R =  -155.049 deg
};
P[2311]{
   GP1:
	UF : 7, UT : 3,	CONFIG : 'F U T, 0, 0, 0',
	X =   -34.169  mm,	Y =   309.326  mm,	Z =     0.000  mm,
	W =  -167.363 deg,	P =    -0.002 deg,	R =  -158.094 deg
};
P[2312]{
   GP1:
	UF : 7, UT : 3,	CONFIG : 'F U T, 0, 0, 0',
	X =   -34.169  mm,	Y =   309.326  mm,	Z =     0.000  mm,
	W =  -167.363 deg,	P =    -0.002 deg,	R =  -158.094 deg
};
P[2313]{
   GP1:
	UF : 7, UT : 3,	CONFIG : 'F U T, 0, 0, 0',
	X =   -34.169  mm,	Y =   309.326  mm,	Z =     0.000  mm,
	W =  -167.363 deg,	P =    -0.002 deg,	R =  -158.094 deg
};
P[2314]{
   GP1:
	UF : 7, UT : 3,	CONFIG : 'F U T, 0, 0, 0',
	X =   -34.169  mm,	Y =   309.326  mm,	Z =     0.000  mm,
	W =  -167.363 deg,	P =    -0.002 deg,	R =  -158.094 deg
};
P[2315]{
   GP1:
	UF : 7, UT : 3,	CONFIG : 'F U T, 0, 0, 0',
	X =    34.169  mm,	Y =   309.326  mm,	Z =     0.000  mm,
	W =  -167.363 deg,	P =     0.001 deg,	R =  -171.797 deg
};
P[2316]{
   GP1:
	UF : 7, UT : 3,	CONFIG : 'F U T, 0, 0, 0',
	X =    34.169  mm,	Y =   309.326  mm,	Z =     0.000  mm,
	W =  -167.363 deg,	P =     0.001 deg,	R =  -171.797 deg
};
P[2317]{
   GP1:
	UF : 7, UT : 3,	CONFIG : 'F U T, 0, 0, 0',
	X =    34.169  mm,	Y =   309.326  mm,	Z =     0.000  mm,
	W =  -167.363 deg,	P =     0.001 deg,	R =  -171.797 deg
};
P[2318]{
   GP1:
	UF : 7, UT : 3,	CONFIG : 'F U T, 0, 0, 0',
	X =    34.169  mm,	Y =   309.326  mm,	Z =     0.000  mm,
	W =  -167.363 deg,	P =     0.001 deg,	R =  -171.797 deg
};
P[2319]{
   GP1:
	UF : 7, UT : 3,	CONFIG : 'F U T, 0, 0, 0',
	X =    53.482  mm,	Y =   306.568  mm,	Z =     0.000  mm,
	W =  -167.363 deg,	P =     0.000 deg,	R =  -174.856 deg
};
P[2320]{
   GP1:
	UF : 7, UT : 3,	CONFIG : 'F U T, 0, 0, 0',
	X =    70.739  mm,	Y =   303.048  mm,	Z =     0.000  mm,
	W =  -167.363 deg,	P =     0.000 deg,	R =  -178.048 deg
};
P[2321]{
   GP1:
	UF : 7, UT : 3,	CONFIG : 'F U T, 0, 0, 0',
	X =    87.613  mm,	Y =   298.610  mm,	Z =     0.000  mm,
	W =  -167.363 deg,	P =    -0.001 deg,	R =   178.718 deg
};
P[2322]{
   GP1:
	UF : 7, UT : 3,	CONFIG : 'F U T, 0, 0, 0',
	X =   103.426  mm,	Y =   293.504  mm,	Z =     0.000  mm,
	W =  -167.363 deg,	P =    -0.001 deg,	R =   175.314 deg
};
P[2323]{
   GP1:
	UF : 7, UT : 3,	CONFIG : 'F U T, 0, 0, 0',
	X =   103.426  mm,	Y =   293.504  mm,	Z =     0.000  mm,
	W =  -167.363 deg,	P =    -0.001 deg,	R =   175.314 deg
};
P[2324]{
   GP1:
	UF : 7, UT : 3,	CONFIG : 'F U T, 0, 0, 0',
	X =   103.426  mm,	Y =   293.504  mm,	Z =     0.000  mm,
	W =  -167.363 deg,	P =    -0.001 deg,	R =   175.314 deg
};
P[2325]{
   GP1:
	UF : 7, UT : 3,	CONFIG : 'F U T, 0, 0, 0',
	X =   103.426  mm,	Y =   293.504  mm,	Z =     0.000  mm,
	W =  -167.363 deg,	P =    -0.001 deg,	R =   175.314 deg
};
P[2326]{
   GP1:
	UF : 7, UT : 3,	CONFIG : 'F U T, 0, 0, 0',
	X =   164.987  mm,	Y =   263.859  mm,	Z =     0.000  mm,
	W =  -167.362 deg,	P =     0.002 deg,	R =   162.852 deg
};
P[2327]{
   GP1:
	UF : 7, UT : 3,	CONFIG : 'F U T, 0, 0, 0',
	X =   164.987  mm,	Y =   263.859  mm,	Z =     0.000  mm,
	W =  -167.362 deg,	P =     0.002 deg,	R =   162.852 deg
};
P[2328]{
   GP1:
	UF : 7, UT : 3,	CONFIG : 'F U T, 0, 0, 0',
	X =   164.987  mm,	Y =   263.859  mm,	Z =     0.000  mm,
	W =  -167.362 deg,	P =     0.002 deg,	R =   162.852 deg
};
P[2329]{
   GP1:
	UF : 7, UT : 3,	CONFIG : 'F U T, 0, 0, 0',
	X =   164.987  mm,	Y =   263.859  mm,	Z =     0.000  mm,
	W =  -167.362 deg,	P =     0.002 deg,	R =   162.852 deg
};
P[2330]{
   GP1:
	UF : 7, UT : 3,	CONFIG : 'F U T, 0, 0, 0',
	X =   180.336  mm,	Y =   253.621  mm,	Z =     0.001  mm,
	W =  -167.363 deg,	P =     0.001 deg,	R =   159.654 deg
};
P[2331]{
   GP1:
	UF : 7, UT : 3,	CONFIG : 'F U T, 0, 0, 0',
	X =   194.365  mm,	Y =   243.027  mm,	Z =     0.001  mm,
	W =  -167.363 deg,	P =     0.000 deg,	R =   156.348 deg
};
P[2332]{
   GP1:
	UF : 7, UT : 3,	CONFIG : 'F U T, 0, 0, 0',
	X =   208.006  mm,	Y =   231.478  mm,	Z =     0.001  mm,
	W =  -167.363 deg,	P =    -0.002 deg,	R =   153.093 deg
};
P[2333]{
   GP1:
	UF : 7, UT : 3,	CONFIG : 'F U T, 0, 0, 0',
	X =   220.529  mm,	Y =   219.561  mm,	Z =     0.000  mm,
	W =  -167.363 deg,	P =    -0.003 deg,	R =   149.730 deg
};
P[2334]{
   GP1:
	UF : 7, UT : 3,	CONFIG : 'F U T, 0, 0, 0',
	X =   220.529  mm,	Y =   219.561  mm,	Z =     0.000  mm,
	W =  -167.363 deg,	P =    -0.003 deg,	R =   149.730 deg
};
P[2335]{
   GP1:
	UF : 7, UT : 3,	CONFIG : 'F U T, 0, 0, 0',
	X =   220.529  mm,	Y =   219.561  mm,	Z =     0.000  mm,
	W =  -167.363 deg,	P =    -0.003 deg,	R =   149.730 deg
};
P[2336]{
   GP1:
	UF : 7, UT : 3,	CONFIG : 'F U T, 0, 0, 0',
	X =   220.529  mm,	Y =   219.561  mm,	Z =     0.000  mm,
	W =  -167.363 deg,	P =    -0.003 deg,	R =   149.730 deg
};
P[2337]{
   GP1:
	UF : 7, UT : 3,	CONFIG : 'F U T, 0, 0, 0',
	X =   263.128  mm,	Y =   166.143  mm,	Z =     0.000  mm,
	W =  -167.362 deg,	P =     0.003 deg,	R =   138.011 deg
};
P[2338]{
   GP1:
	UF : 7, UT : 3,	CONFIG : 'F U T, 0, 0, 0',
	X =   263.128  mm,	Y =   166.143  mm,	Z =     0.000  mm,
	W =  -167.362 deg,	P =     0.003 deg,	R =   138.011 deg
};
P[2339]{
   GP1:
	UF : 7, UT : 3,	CONFIG : 'F U T, 0, 0, 0',
	X =   263.128  mm,	Y =   166.143  mm,	Z =     0.000  mm,
	W =  -167.362 deg,	P =     0.003 deg,	R =   138.011 deg
};
P[2340]{
   GP1:
	UF : 7, UT : 3,	CONFIG : 'F U T, 0, 0, 0',
	X =   263.128  mm,	Y =   166.143  mm,	Z =     0.000  mm,
	W =  -167.362 deg,	P =     0.003 deg,	R =   138.011 deg
};
P[2341]{
   GP1:
	UF : 7, UT : 3,	CONFIG : 'F U T, 0, 0, 0',
	X =   271.387  mm,	Y =   152.293  mm,	Z =     0.001  mm,
	W =  -167.362 deg,	P =     0.002 deg,	R =   134.367 deg
};
P[2342]{
   GP1:
	UF : 7, UT : 3,	CONFIG : 'F U T, 0, 0, 0',
	X =   279.519  mm,	Y =   136.786  mm,	Z =     0.001  mm,
	W =  -167.363 deg,	P =     0.000 deg,	R =   131.108 deg
};
P[2343]{
   GP1:
	UF : 7, UT : 3,	CONFIG : 'F U T, 0, 0, 0',
	X =   286.826  mm,	Y =   120.732  mm,	Z =     0.001  mm,
	W =  -167.363 deg,	P =    -0.001 deg,	R =   127.882 deg
};
P[2344]{
   GP1:
	UF : 7, UT : 3,	CONFIG : 'F U T, 0, 0, 0',
	X =   293.963  mm,	Y =   102.140  mm,	Z =     0.000  mm,
	W =  -167.363 deg,	P =    -0.003 deg,	R =   124.693 deg
};
P[2345]{
   GP1:
	UF : 7, UT : 3,	CONFIG : 'F U T, 0, 0, 0',
	X =   293.963  mm,	Y =   102.140  mm,	Z =     0.000  mm,
	W =  -167.363 deg,	P =    -0.003 deg,	R =   124.693 deg
};
P[2346]{
   GP1:
	UF : 7, UT : 3,	CONFIG : 'F U T, 0, 0, 0',
	X =   293.963  mm,	Y =   102.140  mm,	Z =     0.000  mm,
	W =  -167.363 deg,	P =    -0.003 deg,	R =   124.693 deg
};
P[2347]{
   GP1:
	UF : 7, UT : 3,	CONFIG : 'F U T, 0, 0, 0',
	X =   293.963  mm,	Y =   102.140  mm,	Z =     0.000  mm,
	W =  -167.363 deg,	P =    -0.003 deg,	R =   124.693 deg
};
P[2348]{
   GP1:
	UF : 7, UT : 3,	CONFIG : 'F U T, 0, 0, 0',
	X =   309.165  mm,	Y =    35.521  mm,	Z =     0.000  mm,
	W =  -167.363 deg,	P =     0.001 deg,	R =   111.548 deg
};
P[2349]{
   GP1:
	UF : 7, UT : 3,	CONFIG : 'F U T, 0, 0, 0',
	X =   309.165  mm,	Y =    35.521  mm,	Z =     0.000  mm,
	W =  -167.363 deg,	P =     0.001 deg,	R =   111.548 deg
};
P[2350]{
   GP1:
	UF : 7, UT : 3,	CONFIG : 'F U T, 0, 0, 0',
	X =   309.165  mm,	Y =    35.521  mm,	Z =     0.000  mm,
	W =  -167.363 deg,	P =     0.001 deg,	R =   111.548 deg
};
P[2351]{
   GP1:
	UF : 7, UT : 3,	CONFIG : 'F U T, 0, 0, 0',
	X =   309.165  mm,	Y =    35.521  mm,	Z =     0.000  mm,
	W =  -167.363 deg,	P =     0.001 deg,	R =   111.548 deg
};
P[2352]{
   GP1:
	UF : 7, UT : 3,	CONFIG : 'F U T, 0, 0, 0',
	X =   310.616  mm,	Y =    19.029  mm,	Z =     0.000  mm,
	W =  -167.363 deg,	P =     0.000 deg,	R =   108.513 deg
};
P[2353]{
   GP1:
	UF : 7, UT : 3,	CONFIG : 'F U T, 0, 0, 0',
	X =   311.210  mm,	Y =     0.000  mm,	Z =     0.000  mm,
	W =  -167.364 deg,	P =    -0.001 deg,	R =   105.707 deg
};
P[2354]{
   GP1:
	UF : 7, UT : 3,	CONFIG : 'F U T, 0, 0, 0',
	X =   311.210  mm,	Y =     0.000  mm,	Z =     0.000  mm,
	W =  -167.364 deg,	P =    -0.001 deg,	R =   105.707 deg
};
P[2355]{
   GP1:
	UF : 7, UT : 3,	CONFIG : 'F U T, 0, 0, 0',
	X =   311.210  mm,	Y =     0.000  mm,	Z =     0.000  mm,
	W =  -167.364 deg,	P =    -0.001 deg,	R =   105.707 deg
};
P[2356]{
   GP1:
	UF : 7, UT : 3,	CONFIG : 'F U T, 0, 0, 0',
	X =   311.210  mm,	Y =     0.000  mm,	Z =     0.000  mm,
	W =  -167.364 deg,	P =    -0.001 deg,	R =   105.707 deg
};
P[2357]{
   GP1:
	UF : 7, UT : 3,	CONFIG : 'F U T, 0, 0, 0',
	X =   308.076  mm,	Y =     0.000  mm,	Z =     0.000  mm,
	W =  -167.364 deg,	P =    -0.001 deg,	R =   105.682 deg
};
P[2358]{
   GP1:
	UF : 7, UT : 3,	CONFIG : 'F U T, 0, 0, 0',
	X =   308.076  mm,	Y =     0.000  mm,	Z =     0.000  mm,
	W =  -167.364 deg,	P =    -0.001 deg,	R =   105.682 deg
};
P[2359]{
   GP1:
	UF : 7, UT : 3,	CONFIG : 'F U T, 0, 0, 0',
	X =   308.076  mm,	Y =     0.000  mm,	Z =     0.000  mm,
	W =  -167.364 deg,	P =    -0.001 deg,	R =   105.682 deg
};
P[2360]{
   GP1:
	UF : 7, UT : 3,	CONFIG : 'F U T, 0, 0, 0',
	X =   308.076  mm,	Y =     0.000  mm,	Z =     0.000  mm,
	W =  -167.364 deg,	P =    -0.001 deg,	R =   105.682 deg
};
P[2361]{
   GP1:
	UF : 7, UT : 3,	CONFIG : 'F U T, 0, 0, 0',
	X =   307.417  mm,	Y =    20.005  mm,	Z =     0.000  mm,
	W =  -167.363 deg,	P =     0.000 deg,	R =   108.762 deg
};
P[2362]{
   GP1:
	UF : 7, UT : 3,	CONFIG : 'F U T, 0, 0, 0',
	X =   305.931  mm,	Y =    36.146  mm,	Z =     0.000  mm,
	W =  -167.363 deg,	P =     0.001 deg,	R =   112.156 deg
};
P[2363]{
   GP1:
	UF : 7, UT : 3,	CONFIG : 'F U T, 0, 0, 0',
	X =   305.931  mm,	Y =    36.146  mm,	Z =     0.000  mm,
	W =  -167.363 deg,	P =     0.001 deg,	R =   112.156 deg
};
P[2364]{
   GP1:
	UF : 7, UT : 3,	CONFIG : 'F U T, 0, 0, 0',
	X =   305.931  mm,	Y =    36.146  mm,	Z =     0.000  mm,
	W =  -167.363 deg,	P =     0.001 deg,	R =   112.156 deg
};
P[2365]{
   GP1:
	UF : 7, UT : 3,	CONFIG : 'F U T, 0, 0, 0',
	X =   305.931  mm,	Y =    36.146  mm,	Z =     0.000  mm,
	W =  -167.363 deg,	P =     0.001 deg,	R =   112.156 deg
};
P[2366]{
   GP1:
	UF : 7, UT : 3,	CONFIG : 'F U T, 0, 0, 0',
	X =   291.330  mm,	Y =   100.182  mm,	Z =     0.000  mm,
	W =  -167.363 deg,	P =    -0.003 deg,	R =   124.583 deg
};
P[2367]{
   GP1:
	UF : 7, UT : 3,	CONFIG : 'F U T, 0, 0, 0',
	X =   291.330  mm,	Y =   100.182  mm,	Z =     0.000  mm,
	W =  -167.363 deg,	P =    -0.003 deg,	R =   124.583 deg
};
P[2368]{
   GP1:
	UF : 7, UT : 3,	CONFIG : 'F U T, 0, 0, 0',
	X =   291.330  mm,	Y =   100.182  mm,	Z =     0.000  mm,
	W =  -167.363 deg,	P =    -0.003 deg,	R =   124.583 deg
};
P[2369]{
   GP1:
	UF : 7, UT : 3,	CONFIG : 'F U T, 0, 0, 0',
	X =   291.330  mm,	Y =   100.182  mm,	Z =     0.000  mm,
	W =  -167.363 deg,	P =    -0.003 deg,	R =   124.583 deg
};
P[2370]{
   GP1:
	UF : 7, UT : 3,	CONFIG : 'F U T, 0, 0, 0',
	X =   284.235  mm,	Y =   118.808  mm,	Z =     0.001  mm,
	W =  -167.363 deg,	P =    -0.001 deg,	R =   127.721 deg
};
P[2371]{
   GP1:
	UF : 7, UT : 3,	CONFIG : 'F U T, 0, 0, 0',
	X =   276.940  mm,	Y =   134.927  mm,	Z =     0.001  mm,
	W =  -167.363 deg,	P =     0.000 deg,	R =   131.030 deg
};
P[2372]{
   GP1:
	UF : 7, UT : 3,	CONFIG : 'F U T, 0, 0, 0',
	X =   268.749  mm,	Y =   150.603  mm,	Z =     0.001  mm,
	W =  -167.362 deg,	P =     0.002 deg,	R =   134.342 deg
};
P[2373]{
   GP1:
	UF : 7, UT : 3,	CONFIG : 'F U T, 0, 0, 0',
	X =   259.950  mm,	Y =   165.305  mm,	Z =     0.000  mm,
	W =  -167.361 deg,	P =     0.003 deg,	R =   137.784 deg
};
P[2374]{
   GP1:
	UF : 7, UT : 3,	CONFIG : 'F U T, 0, 0, 0',
	X =   259.950  mm,	Y =   165.305  mm,	Z =     0.000  mm,
	W =  -167.361 deg,	P =     0.003 deg,	R =   137.784 deg
};
P[2375]{
   GP1:
	UF : 7, UT : 3,	CONFIG : 'F U T, 0, 0, 0',
	X =   259.950  mm,	Y =   165.305  mm,	Z =     0.000  mm,
	W =  -167.361 deg,	P =     0.003 deg,	R =   137.784 deg
};
P[2376]{
   GP1:
	UF : 7, UT : 3,	CONFIG : 'F U T, 0, 0, 0',
	X =   259.950  mm,	Y =   165.305  mm,	Z =     0.000  mm,
	W =  -167.361 deg,	P =     0.003 deg,	R =   137.784 deg
};
P[2377]{
   GP1:
	UF : 7, UT : 3,	CONFIG : 'F U T, 0, 0, 0',
	X =   219.006  mm,	Y =   216.652  mm,	Z =     0.000  mm,
	W =  -167.363 deg,	P =    -0.003 deg,	R =   149.847 deg
};
P[2378]{
   GP1:
	UF : 7, UT : 3,	CONFIG : 'F U T, 0, 0, 0',
	X =   219.006  mm,	Y =   216.652  mm,	Z =     0.000  mm,
	W =  -167.363 deg,	P =    -0.003 deg,	R =   149.847 deg
};
P[2379]{
   GP1:
	UF : 7, UT : 3,	CONFIG : 'F U T, 0, 0, 0',
	X =   219.006  mm,	Y =   216.652  mm,	Z =     0.000  mm,
	W =  -167.363 deg,	P =    -0.003 deg,	R =   149.847 deg
};
P[2380]{
   GP1:
	UF : 7, UT : 3,	CONFIG : 'F U T, 0, 0, 0',
	X =   219.006  mm,	Y =   216.652  mm,	Z =     0.000  mm,
	W =  -167.363 deg,	P =    -0.003 deg,	R =   149.847 deg
};
P[2381]{
   GP1:
	UF : 7, UT : 3,	CONFIG : 'F U T, 0, 0, 0',
	X =   206.109  mm,	Y =   228.966  mm,	Z =     0.001  mm,
	W =  -167.363 deg,	P =    -0.002 deg,	R =   153.045 deg
};
P[2382]{
   GP1:
	UF : 7, UT : 3,	CONFIG : 'F U T, 0, 0, 0',
	X =   192.670  mm,	Y =   240.370  mm,	Z =     0.001  mm,
	W =  -167.363 deg,	P =     0.000 deg,	R =   156.285 deg
};
P[2383]{
   GP1:
	UF : 7, UT : 3,	CONFIG : 'F U T, 0, 0, 0',
	X =   178.782  mm,	Y =   250.880  mm,	Z =     0.001  mm,
	W =  -167.362 deg,	P =     0.001 deg,	R =   159.566 deg
};
P[2384]{
   GP1:
	UF : 7, UT : 3,	CONFIG : 'F U T, 0, 0, 0',
	X =   162.492  mm,	Y =   261.729  mm,	Z =     0.000  mm,
	W =  -167.362 deg,	P =     0.002 deg,	R =   162.754 deg
};
P[2385]{
   GP1:
	UF : 7, UT : 3,	CONFIG : 'F U T, 0, 0, 0',
	X =   162.492  mm,	Y =   261.729  mm,	Z =     0.000  mm,
	W =  -167.362 deg,	P =     0.002 deg,	R =   162.754 deg
};
P[2386]{
   GP1:
	UF : 7, UT : 3,	CONFIG : 'F U T, 0, 0, 0',
	X =   162.492  mm,	Y =   261.729  mm,	Z =     0.000  mm,
	W =  -167.362 deg,	P =     0.002 deg,	R =   162.754 deg
};
P[2387]{
   GP1:
	UF : 7, UT : 3,	CONFIG : 'F U T, 0, 0, 0',
	X =   162.492  mm,	Y =   261.729  mm,	Z =     0.000  mm,
	W =  -167.362 deg,	P =     0.002 deg,	R =   162.754 deg
};
P[2388]{
   GP1:
	UF : 7, UT : 3,	CONFIG : 'F U T, 0, 0, 0',
	X =   103.316  mm,	Y =   290.215  mm,	Z =     0.000  mm,
	W =  -167.363 deg,	P =    -0.001 deg,	R =   175.057 deg
};
P[2389]{
   GP1:
	UF : 7, UT : 3,	CONFIG : 'F U T, 0, 0, 0',
	X =   103.316  mm,	Y =   290.215  mm,	Z =     0.000  mm,
	W =  -167.363 deg,	P =    -0.001 deg,	R =   175.057 deg
};
P[2390]{
   GP1:
	UF : 7, UT : 3,	CONFIG : 'F U T, 0, 0, 0',
	X =   103.316  mm,	Y =   290.215  mm,	Z =     0.000  mm,
	W =  -167.363 deg,	P =    -0.001 deg,	R =   175.057 deg
};
P[2391]{
   GP1:
	UF : 7, UT : 3,	CONFIG : 'F U T, 0, 0, 0',
	X =   103.316  mm,	Y =   290.215  mm,	Z =     0.000  mm,
	W =  -167.363 deg,	P =    -0.001 deg,	R =   175.057 deg
};
P[2392]{
   GP1:
	UF : 7, UT : 3,	CONFIG : 'F U T, 0, 0, 0',
	X =    86.904  mm,	Y =   295.550  mm,	Z =     0.000  mm,
	W =  -167.363 deg,	P =    -0.001 deg,	R =   178.687 deg
};
P[2393]{
   GP1:
	UF : 7, UT : 3,	CONFIG : 'F U T, 0, 0, 0',
	X =    69.148  mm,	Y =   300.208  mm,	Z =     0.000  mm,
	W =  -167.363 deg,	P =     0.000 deg,	R =  -177.934 deg
};
P[2394]{
   GP1:
	UF : 7, UT : 3,	CONFIG : 'F U T, 0, 0, 0',
	X =    51.213  mm,	Y =   303.771  mm,	Z =     0.000  mm,
	W =  -167.363 deg,	P =     0.000 deg,	R =  -174.529 deg
};
P[2395]{
   GP1:
	UF : 7, UT : 3,	CONFIG : 'F U T, 0, 0, 0',
	X =    32.839  mm,	Y =   306.310  mm,	Z =     0.000  mm,
	W =  -167.363 deg,	P =     0.001 deg,	R =  -171.182 deg
};
P[2396]{
   GP1:
	UF : 7, UT : 3,	CONFIG : 'F U T, 0, 0, 0',
	X =    32.839  mm,	Y =   306.310  mm,	Z =     0.000  mm,
	W =  -167.363 deg,	P =     0.001 deg,	R =  -171.182 deg
};
P[2397]{
   GP1:
	UF : 7, UT : 3,	CONFIG : 'F U T, 0, 0, 0',
	X =    32.839  mm,	Y =   306.310  mm,	Z =     0.000  mm,
	W =  -167.363 deg,	P =     0.001 deg,	R =  -171.182 deg
};
P[2398]{
   GP1:
	UF : 7, UT : 3,	CONFIG : 'F U T, 0, 0, 0',
	X =    32.839  mm,	Y =   306.310  mm,	Z =     0.000  mm,
	W =  -167.363 deg,	P =     0.001 deg,	R =  -171.182 deg
};
P[2399]{
   GP1:
	UF : 7, UT : 3,	CONFIG : 'F U T, 0, 0, 0',
	X =   -32.839  mm,	Y =   306.310  mm,	Z =     0.000  mm,
	W =  -167.363 deg,	P =    -0.002 deg,	R =  -158.763 deg
};
P[2400]{
   GP1:
	UF : 7, UT : 3,	CONFIG : 'F U T, 0, 0, 0',
	X =   -32.839  mm,	Y =   306.310  mm,	Z =     0.000  mm,
	W =  -167.363 deg,	P =    -0.002 deg,	R =  -158.763 deg
};
P[2401]{
   GP1:
	UF : 7, UT : 3,	CONFIG : 'F U T, 0, 0, 0',
	X =   -32.839  mm,	Y =   306.310  mm,	Z =     0.000  mm,
	W =  -167.363 deg,	P =    -0.002 deg,	R =  -158.763 deg
};
P[2402]{
   GP1:
	UF : 7, UT : 3,	CONFIG : 'F U T, 0, 0, 0',
	X =   -32.839  mm,	Y =   306.310  mm,	Z =     0.000  mm,
	W =  -167.363 deg,	P =    -0.002 deg,	R =  -158.763 deg
};
P[2403]{
   GP1:
	UF : 7, UT : 3,	CONFIG : 'F U T, 0, 0, 0',
	X =   -51.187  mm,	Y =   303.775  mm,	Z =     0.001  mm,
	W =  -167.363 deg,	P =     0.000 deg,	R =  -155.378 deg
};
P[2404]{
   GP1:
	UF : 7, UT : 3,	CONFIG : 'F U T, 0, 0, 0',
	X =   -69.186  mm,	Y =   300.195  mm,	Z =     0.001  mm,
	W =  -167.362 deg,	P =     0.002 deg,	R =  -151.956 deg
};
P[2405]{
   GP1:
	UF : 7, UT : 3,	CONFIG : 'F U T, 0, 0, 0',
	X =   -87.004  mm,	Y =   295.523  mm,	Z =     0.001  mm,
	W =  -167.361 deg,	P =     0.003 deg,	R =  -148.552 deg
};
P[2406]{
   GP1:
	UF : 7, UT : 3,	CONFIG : 'F U T, 0, 0, 0',
	X =  -103.316  mm,	Y =   290.215  mm,	Z =     0.000  mm,
	W =  -167.360 deg,	P =     0.005 deg,	R =  -144.822 deg
};
P[2407]{
   GP1:
	UF : 7, UT : 3,	CONFIG : 'F U T, 0, 0, 0',
	X =  -103.316  mm,	Y =   290.215  mm,	Z =     0.000  mm,
	W =  -167.360 deg,	P =     0.005 deg,	R =  -144.822 deg
};
P[2408]{
   GP1:
	UF : 7, UT : 3,	CONFIG : 'F U T, 0, 0, 0',
	X =  -103.316  mm,	Y =   290.215  mm,	Z =     0.000  mm,
	W =  -167.360 deg,	P =     0.005 deg,	R =  -144.822 deg
};
P[2409]{
   GP1:
	UF : 7, UT : 3,	CONFIG : 'F U T, 0, 0, 0',
	X =  -103.316  mm,	Y =   290.215  mm,	Z =     0.000  mm,
	W =  -167.360 deg,	P =     0.005 deg,	R =  -144.822 deg
};
P[2410]{
   GP1:
	UF : 7, UT : 3,	CONFIG : 'F U T, 0, 0, 0',
	X =  -162.492  mm,	Y =   261.729  mm,	Z =     0.000  mm,
	W =  -167.361 deg,	P =    -0.026 deg,	R =  -132.634 deg
};
P[2411]{
   GP1:
	UF : 7, UT : 3,	CONFIG : 'F U T, 0, 0, 0',
	X =  -162.492  mm,	Y =   261.729  mm,	Z =     0.000  mm,
	W =  -167.361 deg,	P =    -0.026 deg,	R =  -132.634 deg
};
P[2412]{
   GP1:
	UF : 7, UT : 3,	CONFIG : 'F U T, 0, 0, 0',
	X =  -162.492  mm,	Y =   261.729  mm,	Z =     0.000  mm,
	W =  -167.361 deg,	P =    -0.026 deg,	R =  -132.634 deg
};
P[2413]{
   GP1:
	UF : 7, UT : 3,	CONFIG : 'F U T, 0, 0, 0',
	X =  -162.492  mm,	Y =   261.729  mm,	Z =     0.000  mm,
	W =  -167.361 deg,	P =    -0.026 deg,	R =  -132.634 deg
};
P[2414]{
   GP1:
	UF : 7, UT : 3,	CONFIG : 'F U T, 0, 0, 0',
	X =  -179.414  mm,	Y =   250.427  mm,	Z =     0.013  mm,
	W =  -167.351 deg,	P =    -0.029 deg,	R =  -129.307 deg
};
P[2415]{
   GP1:
	UF : 7, UT : 3,	CONFIG : 'F U T, 0, 0, 0',
	X =  -193.911  mm,	Y =   239.382  mm,	Z =     0.025  mm,
	W =  -167.341 deg,	P =    -0.032 deg,	R =  -125.943 deg
};
P[2416]{
   GP1:
	UF : 7, UT : 3,	CONFIG : 'F U T, 0, 0, 0',
	X =  -206.662  mm,	Y =   228.463  mm,	Z =     0.025  mm,
	W =  -167.316 deg,	P =     0.043 deg,	R =  -122.818 deg
};
P[2417]{
   GP1:
	UF : 7, UT : 3,	CONFIG : 'F U T, 0, 0, 0',
	X =  -219.006  mm,	Y =   216.652  mm,	Z =     0.000  mm,
	W =  -167.281 deg,	P =     0.116 deg,	R =  -119.743 deg
};
P[2418]{
   GP1:
	UF : 7, UT : 3,	CONFIG : 'F U T, 0, 0, 0',
	X =  -219.006  mm,	Y =   216.652  mm,	Z =     0.000  mm,
	W =  -167.281 deg,	P =     0.116 deg,	R =  -119.743 deg
};
P[2419]{
   GP1:
	UF : 7, UT : 3,	CONFIG : 'F U T, 0, 0, 0',
	X =  -219.006  mm,	Y =   216.652  mm,	Z =     0.000  mm,
	W =  -167.281 deg,	P =     0.116 deg,	R =  -119.743 deg
};
P[2420]{
   GP1:
	UF : 7, UT : 3,	CONFIG : 'F U T, 0, 0, 0',
	X =  -219.006  mm,	Y =   216.652  mm,	Z =     0.000  mm,
	W =  -167.281 deg,	P =     0.116 deg,	R =  -119.743 deg
};
P[2421]{
   GP1:
	UF : 7, UT : 3,	CONFIG : 'F U T, 0, 0, 0',
	X =  -259.950  mm,	Y =   165.305  mm,	Z =     0.000  mm,
	W =  -167.278 deg,	P =    -0.894 deg,	R =  -107.678 deg
};
P[2422]{
   GP1:
	UF : 7, UT : 3,	CONFIG : 'F U T, 0, 0, 0',
	X =  -259.950  mm,	Y =   165.305  mm,	Z =     0.000  mm,
	W =  -167.278 deg,	P =    -0.894 deg,	R =  -107.678 deg
};
P[2423]{
   GP1:
	UF : 7, UT : 3,	CONFIG : 'F U T, 0, 0, 0',
	X =  -259.950  mm,	Y =   165.305  mm,	Z =     0.000  mm,
	W =  -167.278 deg,	P =    -0.894 deg,	R =  -107.678 deg
};
P[2424]{
   GP1:
	UF : 7, UT : 3,	CONFIG : 'F U T, 0, 0, 0',
	X =  -259.950  mm,	Y =   165.305  mm,	Z =     0.000  mm,
	W =  -167.278 deg,	P =    -0.894 deg,	R =  -107.678 deg
};
P[2425]{
   GP1:
	UF : 7, UT : 3,	CONFIG : 'F U T, 0, 0, 0',
	X =  -268.025  mm,	Y =   151.867  mm,	Z =     0.241  mm,
	W =  -167.849 deg,	P =    -0.672 deg,	R =  -104.537 deg
};
P[2426]{
   GP1:
	UF : 7, UT : 3,	CONFIG : 'F U T, 0, 0, 0',
	X =  -277.242  mm,	Y =   134.307  mm,	Z =     0.372  mm,
	W =  -168.105 deg,	P =     0.277 deg,	R =  -100.816 deg
};
P[2427]{
   GP1:
	UF : 7, UT : 3,	CONFIG : 'F U T, 0, 0, 0',
	X =  -284.120  mm,	Y =   119.090  mm,	Z =     0.239  mm,
	W =  -167.714 deg,	P =     0.904 deg,	R =   -97.675 deg
};
P[2428]{
   GP1:
	UF : 7, UT : 3,	CONFIG : 'F U T, 0, 0, 0',
	X =  -286.488  mm,	Y =   113.262  mm,	Z =     0.148  mm,
	W =  -167.475 deg,	P =     0.882 deg,	R =   -96.516 deg
};
P[2429]{
   GP1:
	UF : 7, UT : 3,	CONFIG : 'F U T, 0, 0, 0',
	X =  -291.330  mm,	Y =   100.182  mm,	Z =     0.000  mm,
	W =  -167.183 deg,	P =     0.258 deg,	R =   -94.472 deg
};
P[2430]{
   GP1:
	UF : 7, UT : 3,	CONFIG : 'F U T, 0, 0, 0',
	X =  -291.330  mm,	Y =   100.182  mm,	Z =     0.000  mm,
	W =  -167.183 deg,	P =     0.258 deg,	R =   -94.472 deg
};
P[2431]{
   GP1:
	UF : 7, UT : 3,	CONFIG : 'F U T, 0, 0, 0',
	X =  -291.330  mm,	Y =   100.182  mm,	Z =     0.000  mm,
	W =  -167.183 deg,	P =     0.258 deg,	R =   -94.472 deg
};
P[2432]{
   GP1:
	UF : 7, UT : 3,	CONFIG : 'F U T, 0, 0, 0',
	X =  -291.330  mm,	Y =   100.182  mm,	Z =     0.000  mm,
	W =  -167.183 deg,	P =     0.258 deg,	R =   -94.472 deg
};
P[2433]{
   GP1:
	UF : 7, UT : 3,	CONFIG : 'F U T, 0, 1, 0',
	X =  -305.931  mm,	Y =    36.146  mm,	Z =     0.000  mm,
	W =  -167.363 deg,	P =    -0.009 deg,	R =   -82.066 deg
};
P[2434]{
   GP1:
	UF : 7, UT : 3,	CONFIG : 'F U T, 0, 1, 0',
	X =  -305.931  mm,	Y =    36.146  mm,	Z =     0.000  mm,
	W =  -167.363 deg,	P =    -0.009 deg,	R =   -82.066 deg
};
P[2435]{
   GP1:
	UF : 7, UT : 3,	CONFIG : 'F U T, 0, 1, 0',
	X =  -305.931  mm,	Y =    36.146  mm,	Z =     0.000  mm,
	W =  -167.363 deg,	P =    -0.009 deg,	R =   -82.066 deg
};
P[2436]{
   GP1:
	UF : 7, UT : 3,	CONFIG : 'F U T, 0, 1, 0',
	X =  -305.931  mm,	Y =    36.146  mm,	Z =     0.000  mm,
	W =  -167.363 deg,	P =    -0.009 deg,	R =   -82.066 deg
};
P[2437]{
   GP1:
	UF : 7, UT : 3,	CONFIG : 'F U T, 0, 1, 0',
	X =  -307.420  mm,	Y =    19.970  mm,	Z =     0.001  mm,
	W =  -167.363 deg,	P =    -0.003 deg,	R =   -78.641 deg
};
P[2438]{
   GP1:
	UF : 7, UT : 3,	CONFIG : 'F U T, 0, 1, 0',
	X =  -308.076  mm,	Y =     0.000  mm,	Z =     0.000  mm,
	W =  -167.362 deg,	P =     0.005 deg,	R =   -75.572 deg
};
P[2439]{
   GP1:
	UF : 7, UT : 3,	CONFIG : 'F U T, 0, 1, 0',
	X =  -308.076  mm,	Y =     0.000  mm,	Z =     0.000  mm,
	W =  -167.362 deg,	P =     0.005 deg,	R =   -75.572 deg
};
P[2440]{
   GP1:
	UF : 7, UT : 3,	CONFIG : 'F U T, 0, 1, 0',
	X =  -308.076  mm,	Y =     0.000  mm,	Z =     0.000  mm,
	W =  -167.362 deg,	P =     0.005 deg,	R =   -75.572 deg
};
P[2441]{
   GP1:
	UF : 7, UT : 3,	CONFIG : 'F U T, 0, 1, 0',
	X =  -308.076  mm,	Y =     0.000  mm,	Z =     0.000  mm,
	W =  -167.362 deg,	P =     0.005 deg,	R =   -75.572 deg
};
P[2442]{
   GP1:
	UF : 7, UT : 3,	CONFIG : 'F U T, 0, 1, 0',
	X =  -304.941  mm,	Y =     0.000  mm,	Z =     0.000  mm,
	W =  -167.362 deg,	P =     0.005 deg,	R =   -75.574 deg
};
P[2443]{
   GP1:
	UF : 7, UT : 3,	CONFIG : 'F U T, 0, 1, 0',
	X =  -304.941  mm,	Y =     0.000  mm,	Z =     0.000  mm,
	W =  -167.362 deg,	P =     0.005 deg,	R =   -75.574 deg
};
P[2444]{
   GP1:
	UF : 7, UT : 3,	CONFIG : 'F U T, 0, 1, 0',
	X =  -304.941  mm,	Y =     0.000  mm,	Z =     0.000  mm,
	W =  -167.362 deg,	P =     0.005 deg,	R =   -75.574 deg
};
P[2445]{
   GP1:
	UF : 7, UT : 3,	CONFIG : 'F U T, 0, 1, 0',
	X =  -304.941  mm,	Y =     0.000  mm,	Z =     0.000  mm,
	W =  -167.362 deg,	P =     0.005 deg,	R =   -75.574 deg
};
P[2446]{
   GP1:
	UF : 7, UT : 3,	CONFIG : 'F U T, 0, 1, 0',
	X =  -304.235  mm,	Y =    20.569  mm,	Z =     0.001  mm,
	W =  -167.362 deg,	P =    -0.003 deg,	R =   -78.821 deg
};
P[2447]{
   GP1:
	UF : 7, UT : 3,	CONFIG : 'F U T, 0, 1, 0',
	X =  -302.657  mm,	Y =    37.100  mm,	Z =     0.000  mm,
	W =  -167.362 deg,	P =    -0.009 deg,	R =   -82.473 deg
};
P[2448]{
   GP1:
	UF : 7, UT : 3,	CONFIG : 'F U T, 0, 1, 0',
	X =  -302.657  mm,	Y =    37.100  mm,	Z =     0.000  mm,
	W =  -167.362 deg,	P =    -0.009 deg,	R =   -82.473 deg
};
P[2449]{
   GP1:
	UF : 7, UT : 3,	CONFIG : 'F U T, 0, 1, 0',
	X =  -302.657  mm,	Y =    37.100  mm,	Z =     0.000  mm,
	W =  -167.362 deg,	P =    -0.009 deg,	R =   -82.473 deg
};
P[2450]{
   GP1:
	UF : 7, UT : 3,	CONFIG : 'F U T, 0, 1, 0',
	X =  -302.657  mm,	Y =    37.100  mm,	Z =     0.000  mm,
	W =  -167.362 deg,	P =    -0.009 deg,	R =   -82.473 deg
};
P[2451]{
   GP1:
	UF : 7, UT : 3,	CONFIG : 'F U T, 0, 0, 0',
	X =  -288.786  mm,	Y =    97.897  mm,	Z =     0.000  mm,
	W =  -167.202 deg,	P =     0.184 deg,	R =   -93.651 deg
};
P[2452]{
   GP1:
	UF : 7, UT : 3,	CONFIG : 'F U T, 0, 0, 0',
	X =  -288.786  mm,	Y =    97.897  mm,	Z =     0.000  mm,
	W =  -167.202 deg,	P =     0.184 deg,	R =   -93.651 deg
};
P[2453]{
   GP1:
	UF : 7, UT : 3,	CONFIG : 'F U T, 0, 0, 0',
	X =  -288.786  mm,	Y =    97.897  mm,	Z =     0.000  mm,
	W =  -167.202 deg,	P =     0.184 deg,	R =   -93.651 deg
};
P[2454]{
   GP1:
	UF : 7, UT : 3,	CONFIG : 'F U T, 0, 0, 0',
	X =  -288.786  mm,	Y =    97.897  mm,	Z =     0.000  mm,
	W =  -167.202 deg,	P =     0.184 deg,	R =   -93.651 deg
};
P[2455]{
   GP1:
	UF : 7, UT : 3,	CONFIG : 'F U T, 0, 0, 0',
	X =  -283.764  mm,	Y =   111.636  mm,	Z =     0.124  mm,
	W =  -167.453 deg,	P =     0.751 deg,	R =   -96.414 deg
};
P[2456]{
   GP1:
	UF : 7, UT : 3,	CONFIG : 'F U T, 0, 0, 0',
	X =  -278.488  mm,	Y =   124.221  mm,	Z =     0.282  mm,
	W =  -167.897 deg,	P =     0.648 deg,	R =   -98.981 deg
};
P[2457]{
   GP1:
	UF : 7, UT : 3,	CONFIG : 'F U T, 0, 0, 0',
	X =  -269.706  mm,	Y =   142.273  mm,	Z =     0.307  mm,
	W =  -168.021 deg,	P =    -0.180 deg,	R =  -102.754 deg
};
P[2458]{
   GP1:
	UF : 7, UT : 3,	CONFIG : 'F U T, 0, 0, 0',
	X =  -260.315  mm,	Y =   158.807  mm,	Z =     0.096  mm,
	W =  -167.464 deg,	P =    -0.805 deg,	R =  -106.340 deg
};
P[2459]{
   GP1:
	UF : 7, UT : 3,	CONFIG : 'F U T, 0, 0, 0',
	X =  -256.595  mm,	Y =   164.745  mm,	Z =     0.000  mm,
	W =  -167.215 deg,	P =    -0.798 deg,	R =  -107.433 deg
};
P[2460]{
   GP1:
	UF : 7, UT : 3,	CONFIG : 'F U T, 0, 0, 0',
	X =  -256.595  mm,	Y =   164.745  mm,	Z =     0.000  mm,
	W =  -167.215 deg,	P =    -0.798 deg,	R =  -107.433 deg
};
P[2461]{
   GP1:
	UF : 7, UT : 3,	CONFIG : 'F U T, 0, 0, 0',
	X =  -256.595  mm,	Y =   164.745  mm,	Z =     0.000  mm,
	W =  -167.215 deg,	P =    -0.798 deg,	R =  -107.433 deg
};
P[2462]{
   GP1:
	UF : 7, UT : 3,	CONFIG : 'F U T, 0, 0, 0',
	X =  -256.595  mm,	Y =   164.745  mm,	Z =     0.000  mm,
	W =  -167.215 deg,	P =    -0.798 deg,	R =  -107.433 deg
};
P[2463]{
   GP1:
	UF : 7, UT : 3,	CONFIG : 'F U T, 0, 0, 0',
	X =  -217.715  mm,	Y =   213.511  mm,	Z =     0.000  mm,
	W =  -167.267 deg,	P =     0.113 deg,	R =  -119.926 deg
};
P[2464]{
   GP1:
	UF : 7, UT : 3,	CONFIG : 'F U T, 0, 0, 0',
	X =  -217.715  mm,	Y =   213.511  mm,	Z =     0.000  mm,
	W =  -167.267 deg,	P =     0.113 deg,	R =  -119.926 deg
};
P[2465]{
   GP1:
	UF : 7, UT : 3,	CONFIG : 'F U T, 0, 0, 0',
	X =  -217.715  mm,	Y =   213.511  mm,	Z =     0.000  mm,
	W =  -167.267 deg,	P =     0.113 deg,	R =  -119.926 deg
};
P[2466]{
   GP1:
	UF : 7, UT : 3,	CONFIG : 'F U T, 0, 0, 0',
	X =  -217.715  mm,	Y =   213.511  mm,	Z =     0.000  mm,
	W =  -167.267 deg,	P =     0.113 deg,	R =  -119.926 deg
};
P[2467]{
   GP1:
	UF : 7, UT : 3,	CONFIG : 'F U T, 0, 0, 0',
	X =  -204.407  mm,	Y =   226.275  mm,	Z =     0.027  mm,
	W =  -167.311 deg,	P =     0.038 deg,	R =  -122.835 deg
};
P[2468]{
   GP1:
	UF : 7, UT : 3,	CONFIG : 'F U T, 0, 0, 0',
	X =  -192.168  mm,	Y =   236.761  mm,	Z =     0.027  mm,
	W =  -167.342 deg,	P =    -0.031 deg,	R =  -125.887 deg
};
P[2469]{
   GP1:
	UF : 7, UT : 3,	CONFIG : 'F U T, 0, 0, 0',
	X =  -176.870  mm,	Y =   248.395  mm,	Z =     0.014  mm,
	W =  -167.350 deg,	P =    -0.029 deg,	R =  -129.496 deg
};
P[2470]{
   GP1:
	UF : 7, UT : 3,	CONFIG : 'F U T, 0, 0, 0',
	X =  -159.710  mm,	Y =   259.766  mm,	Z =     0.000  mm,
	W =  -167.358 deg,	P =    -0.028 deg,	R =  -132.954 deg
};
P[2471]{
   GP1:
	UF : 7, UT : 3,	CONFIG : 'F U T, 0, 0, 0',
	X =  -159.710  mm,	Y =   259.766  mm,	Z =     0.000  mm,
	W =  -167.358 deg,	P =    -0.028 deg,	R =  -132.954 deg
};
P[2472]{
   GP1:
	UF : 7, UT : 3,	CONFIG : 'F U T, 0, 0, 0',
	X =  -159.710  mm,	Y =   259.766  mm,	Z =     0.000  mm,
	W =  -167.358 deg,	P =    -0.028 deg,	R =  -132.954 deg
};
P[2473]{
   GP1:
	UF : 7, UT : 3,	CONFIG : 'F U T, 0, 0, 0',
	X =  -159.710  mm,	Y =   259.766  mm,	Z =     0.000  mm,
	W =  -167.358 deg,	P =    -0.028 deg,	R =  -132.954 deg
};
P[2474]{
   GP1:
	UF : 7, UT : 3,	CONFIG : 'F U T, 0, 0, 0',
	X =  -103.517  mm,	Y =   286.816  mm,	Z =     0.000  mm,
	W =  -167.359 deg,	P =     0.005 deg,	R =  -144.937 deg
};
P[2475]{
   GP1:
	UF : 7, UT : 3,	CONFIG : 'F U T, 0, 0, 0',
	X =  -103.517  mm,	Y =   286.816  mm,	Z =     0.000  mm,
	W =  -167.359 deg,	P =     0.005 deg,	R =  -144.937 deg
};
P[2476]{
   GP1:
	UF : 7, UT : 3,	CONFIG : 'F U T, 0, 0, 0',
	X =  -103.517  mm,	Y =   286.816  mm,	Z =     0.000  mm,
	W =  -167.359 deg,	P =     0.005 deg,	R =  -144.937 deg
};
P[2477]{
   GP1:
	UF : 7, UT : 3,	CONFIG : 'F U T, 0, 0, 0',
	X =  -103.517  mm,	Y =   286.816  mm,	Z =     0.000  mm,
	W =  -167.359 deg,	P =     0.005 deg,	R =  -144.937 deg
};
P[2478]{
   GP1:
	UF : 7, UT : 3,	CONFIG : 'F U T, 0, 0, 0',
	X =   -85.922  mm,	Y =   292.578  mm,	Z =     0.001  mm,
	W =  -167.361 deg,	P =     0.003 deg,	R =  -148.591 deg
};
P[2479]{
   GP1:
	UF : 7, UT : 3,	CONFIG : 'F U T, 0, 0, 0',
	X =   -67.527  mm,	Y =   297.362  mm,	Z =     0.001  mm,
	W =  -167.362 deg,	P =     0.001 deg,	R =  -152.143 deg
};
P[2480]{
   GP1:
	UF : 7, UT : 3,	CONFIG : 'F U T, 0, 0, 0',
	X =   -48.830  mm,	Y =   300.991  mm,	Z =     0.001  mm,
	W =  -167.362 deg,	P =     0.000 deg,	R =  -155.693 deg
};
P[2481]{
   GP1:
	UF : 7, UT : 3,	CONFIG : 'F U T, 0, 0, 0',
	X =   -31.179  mm,	Y =   303.326  mm,	Z =     0.000  mm,
	W =  -167.363 deg,	P =    -0.002 deg,	R =  -159.537 deg
};
P[2482]{
   GP1:
	UF : 7, UT : 3,	CONFIG : 'F U T, 0, 0, 0',
	X =   -31.179  mm,	Y =   303.326  mm,	Z =     0.000  mm,
	W =  -167.363 deg,	P =    -0.002 deg,	R =  -159.537 deg
};
P[2483]{
   GP1:
	UF : 7, UT : 3,	CONFIG : 'F U T, 0, 0, 0',
	X =   -31.179  mm,	Y =   303.326  mm,	Z =     0.000  mm,
	W =  -167.363 deg,	P =    -0.002 deg,	R =  -159.537 deg
};
P[2484]{
   GP1:
	UF : 7, UT : 3,	CONFIG : 'F U T, 0, 0, 0',
	X =   -31.179  mm,	Y =   303.326  mm,	Z =     0.000  mm,
	W =  -167.363 deg,	P =    -0.002 deg,	R =  -159.537 deg
};
P[2485]{
   GP1:
	UF : 7, UT : 3,	CONFIG : 'F U T, 0, 0, 0',
	X =    31.179  mm,	Y =   303.326  mm,	Z =     0.000  mm,
	W =  -167.362 deg,	P =     0.001 deg,	R =  -170.469 deg
};
P[2486]{
   GP1:
	UF : 7, UT : 3,	CONFIG : 'F U T, 0, 0, 0',
	X =    31.179  mm,	Y =   303.326  mm,	Z =     0.000  mm,
	W =  -167.362 deg,	P =     0.001 deg,	R =  -170.469 deg
};
P[2487]{
   GP1:
	UF : 7, UT : 3,	CONFIG : 'F U T, 0, 0, 0',
	X =    31.179  mm,	Y =   303.326  mm,	Z =     0.000  mm,
	W =  -167.362 deg,	P =     0.001 deg,	R =  -170.469 deg
};
P[2488]{
   GP1:
	UF : 7, UT : 3,	CONFIG : 'F U T, 0, 0, 0',
	X =    31.179  mm,	Y =   303.326  mm,	Z =     0.000  mm,
	W =  -167.362 deg,	P =     0.001 deg,	R =  -170.469 deg
};
P[2489]{
   GP1:
	UF : 7, UT : 3,	CONFIG : 'F U T, 0, 0, 0',
	X =    49.048  mm,	Y =   300.955  mm,	Z =     0.000  mm,
	W =  -167.363 deg,	P =     0.001 deg,	R =  -174.225 deg
};
P[2490]{
   GP1:
	UF : 7, UT : 3,	CONFIG : 'F U T, 0, 0, 0',
	X =    67.642  mm,	Y =   297.336  mm,	Z =     0.001  mm,
	W =  -167.363 deg,	P =     0.000 deg,	R =  -177.775 deg
};
P[2491]{
   GP1:
	UF : 7, UT : 3,	CONFIG : 'F U T, 0, 0, 0',
	X =    85.984  mm,	Y =   292.561  mm,	Z =     0.000  mm,
	W =  -167.363 deg,	P =    -0.001 deg,	R =   178.685 deg
};
P[2492]{
   GP1:
	UF : 7, UT : 3,	CONFIG : 'F U T, 0, 0, 0',
	X =   103.517  mm,	Y =   286.816  mm,	Z =     0.000  mm,
	W =  -167.363 deg,	P =    -0.002 deg,	R =   175.040 deg
};
P[2493]{
   GP1:
	UF : 7, UT : 3,	CONFIG : 'F U T, 0, 0, 0',
	X =   103.517  mm,	Y =   286.816  mm,	Z =     0.000  mm,
	W =  -167.363 deg,	P =    -0.002 deg,	R =   175.040 deg
};
P[2494]{
   GP1:
	UF : 7, UT : 3,	CONFIG : 'F U T, 0, 0, 0',
	X =   103.517  mm,	Y =   286.816  mm,	Z =     0.000  mm,
	W =  -167.363 deg,	P =    -0.002 deg,	R =   175.040 deg
};
P[2495]{
   GP1:
	UF : 7, UT : 3,	CONFIG : 'F U T, 0, 0, 0',
	X =   103.517  mm,	Y =   286.816  mm,	Z =     0.000  mm,
	W =  -167.363 deg,	P =    -0.002 deg,	R =   175.040 deg
};
P[2496]{
   GP1:
	UF : 7, UT : 3,	CONFIG : 'F U T, 0, 0, 0',
	X =   159.710  mm,	Y =   259.766  mm,	Z =     0.000  mm,
	W =  -167.361 deg,	P =     0.002 deg,	R =   163.030 deg
};
P[2497]{
   GP1:
	UF : 7, UT : 3,	CONFIG : 'F U T, 0, 0, 0',
	X =   159.710  mm,	Y =   259.766  mm,	Z =     0.000  mm,
	W =  -167.361 deg,	P =     0.002 deg,	R =   163.030 deg
};
P[2498]{
   GP1:
	UF : 7, UT : 3,	CONFIG : 'F U T, 0, 0, 0',
	X =   159.710  mm,	Y =   259.766  mm,	Z =     0.000  mm,
	W =  -167.361 deg,	P =     0.002 deg,	R =   163.030 deg
};
P[2499]{
   GP1:
	UF : 7, UT : 3,	CONFIG : 'F U T, 0, 0, 0',
	X =   159.710  mm,	Y =   259.766  mm,	Z =     0.000  mm,
	W =  -167.361 deg,	P =     0.002 deg,	R =   163.030 deg
};
P[2500]{
   GP1:
	UF : 7, UT : 3,	CONFIG : 'F U T, 0, 0, 0',
	X =   175.767  mm,	Y =   249.174  mm,	Z =     0.001  mm,
	W =  -167.362 deg,	P =     0.001 deg,	R =   159.839 deg
};
P[2501]{
   GP1:
	UF : 7, UT : 3,	CONFIG : 'F U T, 0, 0, 0',
	X =   189.909  mm,	Y =   238.564  mm,	Z =     0.001  mm,
	W =  -167.362 deg,	P =     0.000 deg,	R =   156.522 deg
};
P[2502]{
   GP1:
	UF : 7, UT : 3,	CONFIG : 'F U T, 0, 0, 0',
	X =   203.382  mm,	Y =   227.196  mm,	Z =     0.001  mm,
	W =  -167.363 deg,	P =    -0.002 deg,	R =   153.184 deg
};
P[2503]{
   GP1:
	UF : 7, UT : 3,	CONFIG : 'F U T, 0, 0, 0',
	X =   217.715  mm,	Y =   213.511  mm,	Z =     0.000  mm,
	W =  -167.363 deg,	P =    -0.004 deg,	R =   150.018 deg
};
P[2504]{
   GP1:
	UF : 7, UT : 3,	CONFIG : 'F U T, 0, 0, 0',
	X =   217.715  mm,	Y =   213.511  mm,	Z =     0.000  mm,
	W =  -167.363 deg,	P =    -0.004 deg,	R =   150.018 deg
};
P[2505]{
   GP1:
	UF : 7, UT : 3,	CONFIG : 'F U T, 0, 0, 0',
	X =   217.715  mm,	Y =   213.511  mm,	Z =     0.000  mm,
	W =  -167.363 deg,	P =    -0.004 deg,	R =   150.018 deg
};
P[2506]{
   GP1:
	UF : 7, UT : 3,	CONFIG : 'F U T, 0, 0, 0',
	X =   217.715  mm,	Y =   213.511  mm,	Z =     0.000  mm,
	W =  -167.363 deg,	P =    -0.004 deg,	R =   150.018 deg
};
P[2507]{
   GP1:
	UF : 7, UT : 3,	CONFIG : 'F U T, 0, 0, 0',
	X =   256.595  mm,	Y =   164.745  mm,	Z =     0.000  mm,
	W =  -167.361 deg,	P =     0.003 deg,	R =   137.543 deg
};
P[2508]{
   GP1:
	UF : 7, UT : 3,	CONFIG : 'F U T, 0, 0, 0',
	X =   256.595  mm,	Y =   164.745  mm,	Z =     0.000  mm,
	W =  -167.361 deg,	P =     0.003 deg,	R =   137.543 deg
};
P[2509]{
   GP1:
	UF : 7, UT : 3,	CONFIG : 'F U T, 0, 0, 0',
	X =   256.595  mm,	Y =   164.745  mm,	Z =     0.000  mm,
	W =  -167.361 deg,	P =     0.003 deg,	R =   137.543 deg
};
P[2510]{
   GP1:
	UF : 7, UT : 3,	CONFIG : 'F U T, 0, 0, 0',
	X =   256.595  mm,	Y =   164.745  mm,	Z =     0.000  mm,
	W =  -167.361 deg,	P =     0.003 deg,	R =   137.543 deg
};
P[2511]{
   GP1:
	UF : 7, UT : 3,	CONFIG : 'F U T, 0, 0, 0',
	X =   266.413  mm,	Y =   148.354  mm,	Z =     0.001  mm,
	W =  -167.362 deg,	P =     0.002 deg,	R =   134.168 deg
};
P[2512]{
   GP1:
	UF : 7, UT : 3,	CONFIG : 'F U T, 0, 0, 0',
	X =   274.926  mm,	Y =   131.894  mm,	Z =     0.001  mm,
	W =  -167.362 deg,	P =     0.000 deg,	R =   130.718 deg
};
P[2513]{
   GP1:
	UF : 7, UT : 3,	CONFIG : 'F U T, 0, 0, 0',
	X =   282.311  mm,	Y =   115.232  mm,	Z =     0.001  mm,
	W =  -167.363 deg,	P =    -0.002 deg,	R =   127.212 deg
};
P[2514]{
   GP1:
	UF : 7, UT : 3,	CONFIG : 'F U T, 0, 0, 0',
	X =   288.786  mm,	Y =    97.897  mm,	Z =     0.000  mm,
	W =  -167.363 deg,	P =    -0.003 deg,	R =   123.755 deg
};
P[2515]{
   GP1:
	UF : 7, UT : 3,	CONFIG : 'F U T, 0, 0, 0',
	X =   288.786  mm,	Y =    97.897  mm,	Z =     0.000  mm,
	W =  -167.363 deg,	P =    -0.003 deg,	R =   123.755 deg
};
P[2516]{
   GP1:
	UF : 7, UT : 3,	CONFIG : 'F U T, 0, 0, 0',
	X =   288.786  mm,	Y =    97.897  mm,	Z =     0.000  mm,
	W =  -167.363 deg,	P =    -0.003 deg,	R =   123.755 deg
};
P[2517]{
   GP1:
	UF : 7, UT : 3,	CONFIG : 'F U T, 0, 0, 0',
	X =   288.786  mm,	Y =    97.897  mm,	Z =     0.000  mm,
	W =  -167.363 deg,	P =    -0.003 deg,	R =   123.755 deg
};
P[2518]{
   GP1:
	UF : 7, UT : 3,	CONFIG : 'F U T, 0, 0, 0',
	X =   302.657  mm,	Y =    37.100  mm,	Z =     0.000  mm,
	W =  -167.363 deg,	P =     0.001 deg,	R =   112.699 deg
};
P[2519]{
   GP1:
	UF : 7, UT : 3,	CONFIG : 'F U T, 0, 0, 0',
	X =   302.657  mm,	Y =    37.100  mm,	Z =     0.000  mm,
	W =  -167.363 deg,	P =     0.001 deg,	R =   112.699 deg
};
P[2520]{
   GP1:
	UF : 7, UT : 3,	CONFIG : 'F U T, 0, 0, 0',
	X =   302.657  mm,	Y =    37.100  mm,	Z =     0.000  mm,
	W =  -167.363 deg,	P =     0.001 deg,	R =   112.699 deg
};
P[2521]{
   GP1:
	UF : 7, UT : 3,	CONFIG : 'F U T, 0, 0, 0',
	X =   302.657  mm,	Y =    37.100  mm,	Z =     0.000  mm,
	W =  -167.363 deg,	P =     0.001 deg,	R =   112.699 deg
};
P[2522]{
   GP1:
	UF : 7, UT : 3,	CONFIG : 'F U T, 0, 0, 0',
	X =   304.239  mm,	Y =    20.505  mm,	Z =     0.000  mm,
	W =  -167.363 deg,	P =     0.000 deg,	R =   108.914 deg
};
P[2523]{
   GP1:
	UF : 7, UT : 3,	CONFIG : 'F U T, 0, 0, 0',
	X =   304.941  mm,	Y =     0.000  mm,	Z =     0.000  mm,
	W =  -167.364 deg,	P =    -0.001 deg,	R =   105.666 deg
};
P[2524]{
   GP1:
	UF : 7, UT : 3,	CONFIG : 'F U T, 0, 0, 0',
	X =   304.941  mm,	Y =     0.000  mm,	Z =     0.000  mm,
	W =  -167.364 deg,	P =    -0.001 deg,	R =   105.666 deg
};
P[2525]{
   GP1:
	UF : 7, UT : 3,	CONFIG : 'F U T, 0, 0, 0',
	X =   304.941  mm,	Y =     0.000  mm,	Z =     0.000  mm,
	W =  -167.364 deg,	P =    -0.001 deg,	R =   105.666 deg
};
P[2526]{
   GP1:
	UF : 7, UT : 3,	CONFIG : 'F U T, 0, 0, 0',
	X =   304.941  mm,	Y =     0.000  mm,	Z =     0.000  mm,
	W =  -167.364 deg,	P =    -0.001 deg,	R =   105.666 deg
};
P[2527]{
   GP1:
	UF : 7, UT : 3,	CONFIG : 'F U T, 0, 0, 0',
	X =   301.807  mm,	Y =     0.000  mm,	Z =     0.000  mm,
	W =  -167.364 deg,	P =    -0.001 deg,	R =   105.691 deg
};
P[2528]{
   GP1:
	UF : 7, UT : 3,	CONFIG : 'F U T, 0, 0, 0',
	X =   301.807  mm,	Y =     0.000  mm,	Z =     0.000  mm,
	W =  -167.364 deg,	P =    -0.001 deg,	R =   105.691 deg
};
P[2529]{
   GP1:
	UF : 7, UT : 3,	CONFIG : 'F U T, 0, 0, 0',
	X =   301.807  mm,	Y =     0.000  mm,	Z =     0.000  mm,
	W =  -167.364 deg,	P =    -0.001 deg,	R =   105.691 deg
};
P[2530]{
   GP1:
	UF : 7, UT : 3,	CONFIG : 'F U T, 0, 0, 0',
	X =   301.807  mm,	Y =     0.000  mm,	Z =     0.000  mm,
	W =  -167.364 deg,	P =    -0.001 deg,	R =   105.691 deg
};
P[2531]{
   GP1:
	UF : 7, UT : 3,	CONFIG : 'F U T, 0, 0, 0',
	X =   301.138  mm,	Y =    19.958  mm,	Z =     0.000  mm,
	W =  -167.363 deg,	P =     0.000 deg,	R =   108.841 deg
};
P[2532]{
   GP1:
	UF : 7, UT : 3,	CONFIG : 'F U T, 0, 0, 0',
	X =   299.339  mm,	Y =    38.417  mm,	Z =     0.000  mm,
	W =  -167.362 deg,	P =     0.001 deg,	R =   112.064 deg
};
P[2533]{
   GP1:
	UF : 7, UT : 3,	CONFIG : 'F U T, 0, 0, 0',
	X =   299.339  mm,	Y =    38.417  mm,	Z =     0.000  mm,
	W =  -167.362 deg,	P =     0.001 deg,	R =   112.064 deg
};
P[2534]{
   GP1:
	UF : 7, UT : 3,	CONFIG : 'F U T, 0, 0, 0',
	X =   299.339  mm,	Y =    38.417  mm,	Z =     0.000  mm,
	W =  -167.362 deg,	P =     0.001 deg,	R =   112.064 deg
};
P[2535]{
   GP1:
	UF : 7, UT : 3,	CONFIG : 'F U T, 0, 0, 0',
	X =   299.339  mm,	Y =    38.417  mm,	Z =     0.000  mm,
	W =  -167.362 deg,	P =     0.001 deg,	R =   112.064 deg
};
P[2536]{
   GP1:
	UF : 7, UT : 3,	CONFIG : 'F U T, 0, 0, 0',
	X =   286.360  mm,	Y =    95.261  mm,	Z =     0.000  mm,
	W =  -167.363 deg,	P =    -0.003 deg,	R =   122.961 deg
};
P[2537]{
   GP1:
	UF : 7, UT : 3,	CONFIG : 'F U T, 0, 0, 0',
	X =   286.360  mm,	Y =    95.261  mm,	Z =     0.000  mm,
	W =  -167.363 deg,	P =    -0.003 deg,	R =   122.961 deg
};
P[2538]{
   GP1:
	UF : 7, UT : 3,	CONFIG : 'F U T, 0, 0, 0',
	X =   286.360  mm,	Y =    95.261  mm,	Z =     0.000  mm,
	W =  -167.363 deg,	P =    -0.003 deg,	R =   122.961 deg
};
P[2539]{
   GP1:
	UF : 7, UT : 3,	CONFIG : 'F U T, 0, 0, 0',
	X =   286.360  mm,	Y =    95.261  mm,	Z =     0.000  mm,
	W =  -167.363 deg,	P =    -0.003 deg,	R =   122.961 deg
};
P[2540]{
   GP1:
	UF : 7, UT : 3,	CONFIG : 'F U T, 0, 0, 0',
	X =   280.193  mm,	Y =   112.129  mm,	Z =     0.001  mm,
	W =  -167.362 deg,	P =    -0.002 deg,	R =   126.891 deg
};
P[2541]{
   GP1:
	UF : 7, UT : 3,	CONFIG : 'F U T, 0, 0, 0',
	X =   272.505  mm,	Y =   129.697  mm,	Z =     0.002  mm,
	W =  -167.362 deg,	P =     0.000 deg,	R =   130.518 deg
};
P[2542]{
   GP1:
	UF : 7, UT : 3,	CONFIG : 'F U T, 0, 0, 0',
	X =   263.715  mm,	Y =   146.761  mm,	Z =     0.001  mm,
	W =  -167.361 deg,	P =     0.001 deg,	R =   134.142 deg
};
P[2543]{
   GP1:
	UF : 7, UT : 3,	CONFIG : 'F U T, 0, 0, 0',
	X =   253.037  mm,	Y =   164.491  mm,	Z =     0.000  mm,
	W =  -167.360 deg,	P =     0.003 deg,	R =   137.610 deg
};
P[2544]{
   GP1:
	UF : 7, UT : 3,	CONFIG : 'F U T, 0, 0, 0',
	X =   253.037  mm,	Y =   164.491  mm,	Z =     0.000  mm,
	W =  -167.360 deg,	P =     0.003 deg,	R =   137.610 deg
};
P[2545]{
   GP1:
	UF : 7, UT : 3,	CONFIG : 'F U T, 0, 0, 0',
	X =   253.037  mm,	Y =   164.491  mm,	Z =     0.000  mm,
	W =  -167.360 deg,	P =     0.003 deg,	R =   137.610 deg
};
P[2546]{
   GP1:
	UF : 7, UT : 3,	CONFIG : 'F U T, 0, 0, 0',
	X =   253.037  mm,	Y =   164.491  mm,	Z =     0.000  mm,
	W =  -167.360 deg,	P =     0.003 deg,	R =   137.610 deg
};
P[2547]{
   GP1:
	UF : 7, UT : 3,	CONFIG : 'F U T, 0, 0, 0',
	X =   216.671  mm,	Y =   210.081  mm,	Z =     0.000  mm,
	W =  -167.362 deg,	P =    -0.004 deg,	R =   149.212 deg
};
P[2548]{
   GP1:
	UF : 7, UT : 3,	CONFIG : 'F U T, 0, 0, 0',
	X =   216.671  mm,	Y =   210.081  mm,	Z =     0.000  mm,
	W =  -167.362 deg,	P =    -0.004 deg,	R =   149.212 deg
};
P[2549]{
   GP1:
	UF : 7, UT : 3,	CONFIG : 'F U T, 0, 0, 0',
	X =   216.671  mm,	Y =   210.081  mm,	Z =     0.000  mm,
	W =  -167.362 deg,	P =    -0.004 deg,	R =   149.212 deg
};
P[2550]{
   GP1:
	UF : 7, UT : 3,	CONFIG : 'F U T, 0, 0, 0',
	X =   216.671  mm,	Y =   210.081  mm,	Z =     0.000  mm,
	W =  -167.362 deg,	P =    -0.004 deg,	R =   149.212 deg
};
P[2551]{
   GP1:
	UF : 7, UT : 3,	CONFIG : 'F U T, 0, 0, 0',
	X =   202.652  mm,	Y =   223.633  mm,	Z =     0.001  mm,
	W =  -167.362 deg,	P =    -0.002 deg,	R =   152.893 deg
};
P[2552]{
   GP1:
	UF : 7, UT : 3,	CONFIG : 'F U T, 0, 0, 0',
	X =   187.806  mm,	Y =   236.233  mm,	Z =     0.002  mm,
	W =  -167.362 deg,	P =     0.000 deg,	R =   156.570 deg
};
P[2553]{
   GP1:
	UF : 7, UT : 3,	CONFIG : 'F U T, 0, 0, 0',
	X =   172.183  mm,	Y =   247.853  mm,	Z =     0.001  mm,
	W =  -167.361 deg,	P =     0.001 deg,	R =   160.241 deg
};
P[2554]{
   GP1:
	UF : 7, UT : 3,	CONFIG : 'F U T, 0, 0, 0',
	X =   156.595  mm,	Y =   257.984  mm,	Z =     0.000  mm,
	W =  -167.361 deg,	P =     0.002 deg,	R =   164.120 deg
};
P[2555]{
   GP1:
	UF : 7, UT : 3,	CONFIG : 'F U T, 0, 0, 0',
	X =   156.595  mm,	Y =   257.984  mm,	Z =     0.000  mm,
	W =  -167.361 deg,	P =     0.002 deg,	R =   164.120 deg
};
P[2556]{
   GP1:
	UF : 7, UT : 3,	CONFIG : 'F U T, 0, 0, 0',
	X =   156.595  mm,	Y =   257.984  mm,	Z =     0.000  mm,
	W =  -167.361 deg,	P =     0.002 deg,	R =   164.120 deg
};
P[2557]{
   GP1:
	UF : 7, UT : 3,	CONFIG : 'F U T, 0, 0, 0',
	X =   156.595  mm,	Y =   257.984  mm,	Z =     0.000  mm,
	W =  -167.361 deg,	P =     0.002 deg,	R =   164.120 deg
};
P[2558]{
   GP1:
	UF : 7, UT : 3,	CONFIG : 'F U T, 0, 0, 0',
	X =   104.062  mm,	Y =   283.293  mm,	Z =     0.000  mm,
	W =  -167.363 deg,	P =    -0.002 deg,	R =   175.392 deg
};
P[2559]{
   GP1:
	UF : 7, UT : 3,	CONFIG : 'F U T, 0, 0, 0',
	X =   104.062  mm,	Y =   283.293  mm,	Z =     0.000  mm,
	W =  -167.363 deg,	P =    -0.002 deg,	R =   175.392 deg
};
P[2560]{
   GP1:
	UF : 7, UT : 3,	CONFIG : 'F U T, 0, 0, 0',
	X =   104.062  mm,	Y =   283.293  mm,	Z =     0.000  mm,
	W =  -167.363 deg,	P =    -0.002 deg,	R =   175.392 deg
};
P[2561]{
   GP1:
	UF : 7, UT : 3,	CONFIG : 'F U T, 0, 0, 0',
	X =   104.062  mm,	Y =   283.293  mm,	Z =     0.000  mm,
	W =  -167.363 deg,	P =    -0.002 deg,	R =   175.392 deg
};
P[2562]{
   GP1:
	UF : 7, UT : 3,	CONFIG : 'F U T, 0, 0, 0',
	X =    84.112  mm,	Y =   289.839  mm,	Z =     0.000  mm,
	W =  -167.363 deg,	P =    -0.001 deg,	R =   178.899 deg
};
P[2563]{
   GP1:
	UF : 7, UT : 3,	CONFIG : 'F U T, 0, 0, 0',
	X =    65.839  mm,	Y =   294.527  mm,	Z =     0.001  mm,
	W =  -167.363 deg,	P =     0.000 deg,	R =  -177.533 deg
};
P[2564]{
   GP1:
	UF : 7, UT : 3,	CONFIG : 'F U T, 0, 0, 0',
	X =    47.299  mm,	Y =   298.070  mm,	Z =     0.000  mm,
	W =  -167.362 deg,	P =     0.001 deg,	R =  -173.969 deg
};
P[2565]{
   GP1:
	UF : 7, UT : 3,	CONFIG : 'F U T, 0, 0, 0',
	X =    29.152  mm,	Y =   300.379  mm,	Z =     0.000  mm,
	W =  -167.362 deg,	P =     0.001 deg,	R =  -170.278 deg
};
P[2566]{
   GP1:
	UF : 7, UT : 3,	CONFIG : 'F U T, 0, 0, 0',
	X =    29.152  mm,	Y =   300.379  mm,	Z =     0.000  mm,
	W =  -167.362 deg,	P =     0.001 deg,	R =  -170.278 deg
};
P[2567]{
   GP1:
	UF : 7, UT : 3,	CONFIG : 'F U T, 0, 0, 0',
	X =    29.152  mm,	Y =   300.379  mm,	Z =     0.000  mm,
	W =  -167.362 deg,	P =     0.001 deg,	R =  -170.278 deg
};
P[2568]{
   GP1:
	UF : 7, UT : 3,	CONFIG : 'F U T, 0, 0, 0',
	X =    29.152  mm,	Y =   300.379  mm,	Z =     0.000  mm,
	W =  -167.362 deg,	P =     0.001 deg,	R =  -170.278 deg
};
P[2569]{
   GP1:
	UF : 7, UT : 3,	CONFIG : 'F U T, 0, 0, 0',
	X =   -29.152  mm,	Y =   300.379  mm,	Z =     0.000  mm,
	W =  -167.363 deg,	P =    -0.003 deg,	R =  -159.616 deg
};
P[2570]{
   GP1:
	UF : 7, UT : 3,	CONFIG : 'F U T, 0, 0, 0',
	X =   -29.152  mm,	Y =   300.379  mm,	Z =     0.000  mm,
	W =  -167.363 deg,	P =    -0.003 deg,	R =  -159.616 deg
};
P[2571]{
   GP1:
	UF : 7, UT : 3,	CONFIG : 'F U T, 0, 0, 0',
	X =   -29.152  mm,	Y =   300.379  mm,	Z =     0.000  mm,
	W =  -167.363 deg,	P =    -0.003 deg,	R =  -159.616 deg
};
P[2572]{
   GP1:
	UF : 7, UT : 3,	CONFIG : 'F U T, 0, 0, 0',
	X =   -29.152  mm,	Y =   300.379  mm,	Z =     0.000  mm,
	W =  -167.363 deg,	P =    -0.003 deg,	R =  -159.616 deg
};
P[2573]{
   GP1:
	UF : 7, UT : 3,	CONFIG : 'F U T, 0, 0, 0',
	X =   -47.299  mm,	Y =   298.070  mm,	Z =     0.001  mm,
	W =  -167.362 deg,	P =    -0.001 deg,	R =  -155.926 deg
};
P[2574]{
   GP1:
	UF : 7, UT : 3,	CONFIG : 'F U T, 0, 0, 0',
	X =   -65.840  mm,	Y =   294.527  mm,	Z =     0.002  mm,
	W =  -167.361 deg,	P =     0.001 deg,	R =  -152.357 deg
};
P[2575]{
   GP1:
	UF : 7, UT : 3,	CONFIG : 'F U T, 0, 0, 0',
	X =   -84.112  mm,	Y =   289.838  mm,	Z =     0.001  mm,
	W =  -167.360 deg,	P =     0.003 deg,	R =  -148.788 deg
};
P[2576]{
   GP1:
	UF : 7, UT : 3,	CONFIG : 'F U T, 0, 0, 0',
	X =  -104.062  mm,	Y =   283.293  mm,	Z =     0.000  mm,
	W =  -167.358 deg,	P =     0.005 deg,	R =  -145.284 deg
};
P[2577]{
   GP1:
	UF : 7, UT : 3,	CONFIG : 'F U T, 0, 0, 0',
	X =  -104.062  mm,	Y =   283.293  mm,	Z =     0.000  mm,
	W =  -167.358 deg,	P =     0.005 deg,	R =  -145.284 deg
};
P[2578]{
   GP1:
	UF : 7, UT : 3,	CONFIG : 'F U T, 0, 0, 0',
	X =  -104.062  mm,	Y =   283.293  mm,	Z =     0.000  mm,
	W =  -167.358 deg,	P =     0.005 deg,	R =  -145.284 deg
};
P[2579]{
   GP1:
	UF : 7, UT : 3,	CONFIG : 'F U T, 0, 0, 0',
	X =  -104.062  mm,	Y =   283.293  mm,	Z =     0.000  mm,
	W =  -167.358 deg,	P =     0.005 deg,	R =  -145.284 deg
};
P[2580]{
   GP1:
	UF : 7, UT : 3,	CONFIG : 'F U T, 0, 0, 0',
	X =  -156.595  mm,	Y =   257.984  mm,	Z =     0.000  mm,
	W =  -167.354 deg,	P =    -0.029 deg,	R =  -134.161 deg
};
P[2581]{
   GP1:
	UF : 7, UT : 3,	CONFIG : 'F U T, 0, 0, 0',
	X =  -156.595  mm,	Y =   257.984  mm,	Z =     0.000  mm,
	W =  -167.354 deg,	P =    -0.029 deg,	R =  -134.161 deg
};
P[2582]{
   GP1:
	UF : 7, UT : 3,	CONFIG : 'F U T, 0, 0, 0',
	X =  -156.595  mm,	Y =   257.984  mm,	Z =     0.000  mm,
	W =  -167.354 deg,	P =    -0.029 deg,	R =  -134.161 deg
};
P[2583]{
   GP1:
	UF : 7, UT : 3,	CONFIG : 'F U T, 0, 0, 0',
	X =  -156.595  mm,	Y =   257.984  mm,	Z =     0.000  mm,
	W =  -167.354 deg,	P =    -0.029 deg,	R =  -134.161 deg
};
P[2584]{
   GP1:
	UF : 7, UT : 3,	CONFIG : 'F U T, 0, 0, 0',
	X =  -173.393  mm,	Y =   247.010  mm,	Z =     0.014  mm,
	W =  -167.350 deg,	P =    -0.029 deg,	R =  -129.898 deg
};
P[2585]{
   GP1:
	UF : 7, UT : 3,	CONFIG : 'F U T, 0, 0, 0',
	X =  -190.194  mm,	Y =   234.325  mm,	Z =     0.029  mm,
	W =  -167.345 deg,	P =    -0.030 deg,	R =  -125.893 deg
};
P[2586]{
   GP1:
	UF : 7, UT : 3,	CONFIG : 'F U T, 0, 0, 0',
	X =  -203.818  mm,	Y =   222.564  mm,	Z =     0.027  mm,
	W =  -167.302 deg,	P =     0.041 deg,	R =  -122.503 deg
};
P[2587]{
   GP1:
	UF : 7, UT : 3,	CONFIG : 'F U T, 0, 0, 0',
	X =  -216.671  mm,	Y =   210.081  mm,	Z =     0.000  mm,
	W =  -167.250 deg,	P =     0.106 deg,	R =  -119.100 deg
};
P[2588]{
   GP1:
	UF : 7, UT : 3,	CONFIG : 'F U T, 0, 0, 0',
	X =  -216.671  mm,	Y =   210.081  mm,	Z =     0.000  mm,
	W =  -167.250 deg,	P =     0.106 deg,	R =  -119.100 deg
};
P[2589]{
   GP1:
	UF : 7, UT : 3,	CONFIG : 'F U T, 0, 0, 0',
	X =  -216.671  mm,	Y =   210.081  mm,	Z =     0.000  mm,
	W =  -167.250 deg,	P =     0.106 deg,	R =  -119.100 deg
};
P[2590]{
   GP1:
	UF : 7, UT : 3,	CONFIG : 'F U T, 0, 0, 0',
	X =  -216.671  mm,	Y =   210.081  mm,	Z =     0.000  mm,
	W =  -167.250 deg,	P =     0.106 deg,	R =  -119.100 deg
};
P[2591]{
   GP1:
	UF : 7, UT : 3,	CONFIG : 'F U T, 0, 0, 0',
	X =  -253.037  mm,	Y =   164.491  mm,	Z =     0.000  mm,
	W =  -167.162 deg,	P =    -0.694 deg,	R =  -107.505 deg
};
P[2592]{
   GP1:
	UF : 7, UT : 3,	CONFIG : 'F U T, 0, 0, 0',
	X =  -253.037  mm,	Y =   164.491  mm,	Z =     0.000  mm,
	W =  -167.162 deg,	P =    -0.694 deg,	R =  -107.505 deg
};
P[2593]{
   GP1:
	UF : 7, UT : 3,	CONFIG : 'F U T, 0, 0, 0',
	X =  -253.037  mm,	Y =   164.491  mm,	Z =     0.000  mm,
	W =  -167.162 deg,	P =    -0.694 deg,	R =  -107.505 deg
};
P[2594]{
   GP1:
	UF : 7, UT : 3,	CONFIG : 'F U T, 0, 0, 0',
	X =  -253.037  mm,	Y =   164.491  mm,	Z =     0.000  mm,
	W =  -167.162 deg,	P =    -0.694 deg,	R =  -107.505 deg
};
P[2595]{
   GP1:
	UF : 7, UT : 3,	CONFIG : 'F U T, 0, 0, 0',
	X =  -261.926  mm,	Y =   149.907  mm,	Z =     0.196  mm,
	W =  -167.750 deg,	P =    -0.491 deg,	R =  -104.769 deg
};
P[2596]{
   GP1:
	UF : 7, UT : 3,	CONFIG : 'F U T, 0, 0, 0',
	X =  -271.252  mm,	Y =   132.292  mm,	Z =     0.292  mm,
	W =  -168.006 deg,	P =     0.249 deg,	R =  -100.949 deg
};
P[2597]{
   GP1:
	UF : 7, UT : 3,	CONFIG : 'F U T, 0, 0, 0',
	X =  -278.311  mm,	Y =   116.729  mm,	Z =     0.182  mm,
	W =  -167.662 deg,	P =     0.704 deg,	R =   -97.694 deg
};
P[2598]{
   GP1:
	UF : 7, UT : 3,	CONFIG : 'F U T, 0, 0, 0',
	X =  -283.687  mm,	Y =   102.971  mm,	Z =     0.038  mm,
	W =  -167.267 deg,	P =     0.382 deg,	R =   -94.885 deg
};
P[2599]{
   GP1:
	UF : 7, UT : 3,	CONFIG : 'F U T, 0, 0, 0',
	X =  -286.360  mm,	Y =    95.261  mm,	Z =     0.000  mm,
	W =  -167.226 deg,	P =     0.128 deg,	R =   -92.852 deg
};
P[2600]{
   GP1:
	UF : 7, UT : 3,	CONFIG : 'F U T, 0, 0, 0',
	X =  -286.360  mm,	Y =    95.261  mm,	Z =     0.000  mm,
	W =  -167.226 deg,	P =     0.128 deg,	R =   -92.852 deg
};
P[2601]{
   GP1:
	UF : 7, UT : 3,	CONFIG : 'F U T, 0, 0, 0',
	X =  -286.360  mm,	Y =    95.261  mm,	Z =     0.000  mm,
	W =  -167.226 deg,	P =     0.128 deg,	R =   -92.852 deg
};
P[2602]{
   GP1:
	UF : 7, UT : 3,	CONFIG : 'F U T, 0, 0, 0',
	X =  -286.360  mm,	Y =    95.261  mm,	Z =     0.000  mm,
	W =  -167.226 deg,	P =     0.128 deg,	R =   -92.852 deg
};
P[2603]{
   GP1:
	UF : 7, UT : 3,	CONFIG : 'F U T, 0, 1, 0',
	X =  -299.339  mm,	Y =    38.417  mm,	Z =     0.000  mm,
	W =  -167.361 deg,	P =    -0.009 deg,	R =   -81.973 deg
};
P[2604]{
   GP1:
	UF : 7, UT : 3,	CONFIG : 'F U T, 0, 1, 0',
	X =  -299.339  mm,	Y =    38.417  mm,	Z =     0.000  mm,
	W =  -167.361 deg,	P =    -0.009 deg,	R =   -81.973 deg
};
P[2605]{
   GP1:
	UF : 7, UT : 3,	CONFIG : 'F U T, 0, 1, 0',
	X =  -299.339  mm,	Y =    38.417  mm,	Z =     0.000  mm,
	W =  -167.361 deg,	P =    -0.009 deg,	R =   -81.973 deg
};
P[2606]{
   GP1:
	UF : 7, UT : 3,	CONFIG : 'F U T, 0, 1, 0',
	X =  -299.339  mm,	Y =    38.417  mm,	Z =     0.000  mm,
	W =  -167.361 deg,	P =    -0.009 deg,	R =   -81.973 deg
};
P[2607]{
   GP1:
	UF : 7, UT : 3,	CONFIG : 'F U T, 0, 1, 0',
	X =  -301.136  mm,	Y =    19.986  mm,	Z =     0.001  mm,
	W =  -167.362 deg,	P =    -0.002 deg,	R =   -78.741 deg
};
P[2608]{
   GP1:
	UF : 7, UT : 3,	CONFIG : 'F U T, 0, 1, 0',
	X =  -301.807  mm,	Y =     0.000  mm,	Z =     0.000  mm,
	W =  -167.362 deg,	P =     0.005 deg,	R =   -75.586 deg
};
P[2609]{
   GP1:
	UF : 7, UT : 3,	CONFIG : 'F U T, 0, 1, 0',
	X =  -301.807  mm,	Y =     0.000  mm,	Z =     0.000  mm,
	W =  -167.362 deg,	P =     0.005 deg,	R =   -75.586 deg
};
P[2610]{
   GP1:
	UF : 7, UT : 3,	CONFIG : 'F U T, 0, 1, 0',
	X =  -301.807  mm,	Y =     0.000  mm,	Z =     0.000  mm,
	W =  -167.362 deg,	P =     0.005 deg,	R =   -75.586 deg
};
P[2611]{
   GP1:
	UF : 7, UT : 3,	CONFIG : 'F U T, 0, 1, 0',
	X =  -301.807  mm,	Y =     0.000  mm,	Z =     0.000  mm,
	W =  -167.362 deg,	P =     0.005 deg,	R =   -75.586 deg
};
P[2612]{
   GP1:
	UF : 7, UT : 3,	CONFIG : 'F U T, 0, 1, 0',
	X =  -298.673  mm,	Y =     0.000  mm,	Z =     0.000  mm,
	W =  -167.362 deg,	P =     0.005 deg,	R =   -75.598 deg
};
P[2613]{
   GP1:
	UF : 7, UT : 3,	CONFIG : 'F U T, 0, 1, 0',
	X =  -298.673  mm,	Y =     0.000  mm,	Z =     0.000  mm,
	W =  -167.362 deg,	P =     0.005 deg,	R =   -75.598 deg
};
P[2614]{
   GP1:
	UF : 7, UT : 3,	CONFIG : 'F U T, 0, 1, 0',
	X =  -298.673  mm,	Y =     0.000  mm,	Z =     0.000  mm,
	W =  -167.362 deg,	P =     0.005 deg,	R =   -75.598 deg
};
P[2615]{
   GP1:
	UF : 7, UT : 3,	CONFIG : 'F U T, 0, 1, 0',
	X =  -298.673  mm,	Y =     0.000  mm,	Z =     0.000  mm,
	W =  -167.362 deg,	P =     0.005 deg,	R =   -75.598 deg
};
P[2616]{
   GP1:
	UF : 7, UT : 3,	CONFIG : 'F U T, 0, 1, 0',
	X =  -297.941  mm,	Y =    20.812  mm,	Z =     0.001  mm,
	W =  -167.361 deg,	P =    -0.003 deg,	R =   -78.951 deg
};
P[2617]{
   GP1:
	UF : 7, UT : 3,	CONFIG : 'F U T, 0, 1, 0',
	X =  -295.952  mm,	Y =    40.176  mm,	Z =     0.000  mm,
	W =  -167.360 deg,	P =    -0.009 deg,	R =   -82.357 deg
};
P[2618]{
   GP1:
	UF : 7, UT : 3,	CONFIG : 'F U T, 0, 1, 0',
	X =  -295.952  mm,	Y =    40.176  mm,	Z =     0.000  mm,
	W =  -167.360 deg,	P =    -0.009 deg,	R =   -82.357 deg
};
P[2619]{
   GP1:
	UF : 7, UT : 3,	CONFIG : 'F U T, 0, 1, 0',
	X =  -295.952  mm,	Y =    40.176  mm,	Z =     0.000  mm,
	W =  -167.360 deg,	P =    -0.009 deg,	R =   -82.357 deg
};
P[2620]{
   GP1:
	UF : 7, UT : 3,	CONFIG : 'F U T, 0, 1, 0',
	X =  -295.952  mm,	Y =    40.176  mm,	Z =     0.000  mm,
	W =  -167.360 deg,	P =    -0.009 deg,	R =   -82.357 deg
};
P[2621]{
   GP1:
	UF : 7, UT : 3,	CONFIG : 'F U T, 0, 0, 0',
	X =  -284.072  mm,	Y =    92.207  mm,	Z =     0.000  mm,
	W =  -167.252 deg,	P =     0.085 deg,	R =   -93.164 deg
};
P[2622]{
   GP1:
	UF : 7, UT : 3,	CONFIG : 'F U T, 0, 0, 0',
	X =  -284.072  mm,	Y =    92.207  mm,	Z =     0.000  mm,
	W =  -167.252 deg,	P =     0.085 deg,	R =   -93.164 deg
};
P[2623]{
   GP1:
	UF : 7, UT : 3,	CONFIG : 'F U T, 0, 0, 0',
	X =  -284.072  mm,	Y =    92.207  mm,	Z =     0.000  mm,
	W =  -167.252 deg,	P =     0.085 deg,	R =   -93.164 deg
};
P[2624]{
   GP1:
	UF : 7, UT : 3,	CONFIG : 'F U T, 0, 0, 0',
	X =  -284.072  mm,	Y =    92.207  mm,	Z =     0.000  mm,
	W =  -167.252 deg,	P =     0.085 deg,	R =   -93.164 deg
};
P[2625]{
   GP1:
	UF : 7, UT : 3,	CONFIG : 'F U T, 0, 0, 0',
	X =  -277.977  mm,	Y =   109.239  mm,	Z =     0.096  mm,
	W =  -167.450 deg,	P =     0.540 deg,	R =   -96.393 deg
};
P[2626]{
   GP1:
	UF : 7, UT : 3,	CONFIG : 'F U T, 0, 0, 0',
	X =  -272.270  mm,	Y =   122.748  mm,	Z =     0.221  mm,
	W =  -167.842 deg,	P =     0.503 deg,	R =   -99.224 deg
};
P[2627]{
   GP1:
	UF : 7, UT : 3,	CONFIG : 'F U T, 0, 0, 0',
	X =  -263.394  mm,	Y =   140.797  mm,	Z =     0.238  mm,
	W =  -167.922 deg,	P =    -0.122 deg,	R =  -103.086 deg
};
P[2628]{
   GP1:
	UF : 7, UT : 3,	CONFIG : 'F U T, 0, 0, 0',
	X =  -253.193  mm,	Y =   158.403  mm,	Z =     0.071  mm,
	W =  -167.353 deg,	P =    -0.605 deg,	R =  -106.999 deg
};
P[2629]{
   GP1:
	UF : 7, UT : 3,	CONFIG : 'F U T, 0, 0, 0',
	X =  -249.198  mm,	Y =   164.607  mm,	Z =     0.000  mm,
	W =  -167.111 deg,	P =    -0.578 deg,	R =  -108.834 deg
};
P[2630]{
   GP1:
	UF : 7, UT : 3,	CONFIG : 'F U T, 0, 0, 0',
	X =  -249.198  mm,	Y =   164.607  mm,	Z =     0.000  mm,
	W =  -167.111 deg,	P =    -0.578 deg,	R =  -108.834 deg
};
P[2631]{
   GP1:
	UF : 7, UT : 3,	CONFIG : 'F U T, 0, 0, 0',
	X =  -249.198  mm,	Y =   164.607  mm,	Z =     0.000  mm,
	W =  -167.111 deg,	P =    -0.578 deg,	R =  -108.834 deg
};
P[2632]{
   GP1:
	UF : 7, UT : 3,	CONFIG : 'F U T, 0, 0, 0',
	X =  -249.198  mm,	Y =   164.607  mm,	Z =     0.000  mm,
	W =  -167.111 deg,	P =    -0.578 deg,	R =  -108.834 deg
};
P[2633]{
   GP1:
	UF : 7, UT : 3,	CONFIG : 'F U T, 0, 0, 0',
	X =  -215.932  mm,	Y =   206.321  mm,	Z =     0.000  mm,
	W =  -167.233 deg,	P =     0.096 deg,	R =  -118.209 deg
};
P[2634]{
   GP1:
	UF : 7, UT : 3,	CONFIG : 'F U T, 0, 0, 0',
	X =  -215.932  mm,	Y =   206.321  mm,	Z =     0.000  mm,
	W =  -167.233 deg,	P =     0.096 deg,	R =  -118.209 deg
};
P[2635]{
   GP1:
	UF : 7, UT : 3,	CONFIG : 'F U T, 0, 0, 0',
	X =  -215.932  mm,	Y =   206.321  mm,	Z =     0.000  mm,
	W =  -167.233 deg,	P =     0.096 deg,	R =  -118.209 deg
};
P[2636]{
   GP1:
	UF : 7, UT : 3,	CONFIG : 'F U T, 0, 0, 0',
	X =  -215.932  mm,	Y =   206.321  mm,	Z =     0.000  mm,
	W =  -167.233 deg,	P =     0.096 deg,	R =  -118.209 deg
};
P[2637]{
   GP1:
	UF : 7, UT : 3,	CONFIG : 'F U T, 0, 0, 0',
	X =  -203.708  mm,	Y =   218.405  mm,	Z =     0.026  mm,
	W =  -167.294 deg,	P =     0.043 deg,	R =  -121.941 deg
};
P[2638]{
   GP1:
	UF : 7, UT : 3,	CONFIG : 'F U T, 0, 0, 0',
	X =  -190.031  mm,	Y =   230.404  mm,	Z =     0.031  mm,
	W =  -167.349 deg,	P =    -0.021 deg,	R =  -125.425 deg
};
P[2639]{
   GP1:
	UF : 7, UT : 3,	CONFIG : 'F U T, 0, 0, 0',
	X =  -178.085  mm,	Y =   239.767  mm,	Z =     0.022  mm,
	W =  -167.350 deg,	P =    -0.024 deg,	R =  -128.356 deg
};
P[2640]{
   GP1:
	UF : 7, UT : 3,	CONFIG : 'F U T, 0, 0, 0',
	X =  -165.638  mm,	Y =   248.516  mm,	Z =     0.009  mm,
	W =  -167.351 deg,	P =    -0.026 deg,	R =  -131.281 deg
};
P[2641]{
   GP1:
	UF : 7, UT : 3,	CONFIG : 'F U T, 0, 0, 0',
	X =  -153.101  mm,	Y =   256.429  mm,	Z =     0.000  mm,
	W =  -167.351 deg,	P =    -0.029 deg,	R =  -134.290 deg
};
P[2642]{
   GP1:
	UF : 7, UT : 3,	CONFIG : 'F U T, 0, 0, 0',
	X =  -153.101  mm,	Y =   256.429  mm,	Z =     0.000  mm,
	W =  -167.351 deg,	P =    -0.029 deg,	R =  -134.290 deg
};
P[2643]{
   GP1:
	UF : 7, UT : 3,	CONFIG : 'F U T, 0, 0, 0',
	X =  -153.101  mm,	Y =   256.429  mm,	Z =     0.000  mm,
	W =  -167.351 deg,	P =    -0.029 deg,	R =  -134.290 deg
};
P[2644]{
   GP1:
	UF : 7, UT : 3,	CONFIG : 'F U T, 0, 0, 0',
	X =  -153.101  mm,	Y =   256.429  mm,	Z =     0.000  mm,
	W =  -167.351 deg,	P =    -0.029 deg,	R =  -134.290 deg
};
P[2645]{
   GP1:
	UF : 7, UT : 3,	CONFIG : 'F U T, 0, 0, 0',
	X =  -105.027  mm,	Y =   279.584  mm,	Z =     0.000  mm,
	W =  -167.357 deg,	P =     0.005 deg,	R =  -144.342 deg
};
P[2646]{
   GP1:
	UF : 7, UT : 3,	CONFIG : 'F U T, 0, 0, 0',
	X =  -105.027  mm,	Y =   279.584  mm,	Z =     0.000  mm,
	W =  -167.357 deg,	P =     0.005 deg,	R =  -144.342 deg
};
P[2647]{
   GP1:
	UF : 7, UT : 3,	CONFIG : 'F U T, 0, 0, 0',
	X =  -105.027  mm,	Y =   279.584  mm,	Z =     0.000  mm,
	W =  -167.357 deg,	P =     0.005 deg,	R =  -144.342 deg
};
P[2648]{
   GP1:
	UF : 7, UT : 3,	CONFIG : 'F U T, 0, 0, 0',
	X =  -105.027  mm,	Y =   279.584  mm,	Z =     0.000  mm,
	W =  -167.357 deg,	P =     0.005 deg,	R =  -144.342 deg
};
P[2649]{
   GP1:
	UF : 7, UT : 3,	CONFIG : 'F U T, 0, 0, 0',
	X =   -86.559  mm,	Y =   285.839  mm,	Z =     0.002  mm,
	W =  -167.359 deg,	P =     0.003 deg,	R =  -148.083 deg
};
P[2650]{
   GP1:
	UF : 7, UT : 3,	CONFIG : 'F U T, 0, 0, 0',
	X =   -67.803  mm,	Y =   290.862  mm,	Z =     0.002  mm,
	W =  -167.360 deg,	P =     0.001 deg,	R =  -151.838 deg
};
P[2651]{
   GP1:
	UF : 7, UT : 3,	CONFIG : 'F U T, 0, 0, 0',
	X =   -48.590  mm,	Y =   294.678  mm,	Z =     0.001  mm,
	W =  -167.361 deg,	P =    -0.001 deg,	R =  -155.563 deg
};
P[2652]{
   GP1:
	UF : 7, UT : 3,	CONFIG : 'F U T, 0, 0, 0',
	X =   -26.690  mm,	Y =   297.475  mm,	Z =     0.000  mm,
	W =  -167.362 deg,	P =    -0.003 deg,	R =  -159.248 deg
};
P[2653]{
   GP1:
	UF : 7, UT : 3,	CONFIG : 'F U T, 0, 0, 0',
	X =   -26.690  mm,	Y =   297.475  mm,	Z =     0.000  mm,
	W =  -167.362 deg,	P =    -0.003 deg,	R =  -159.248 deg
};
P[2654]{
   GP1:
	UF : 7, UT : 3,	CONFIG : 'F U T, 0, 0, 0',
	X =   -26.690  mm,	Y =   297.475  mm,	Z =     0.000  mm,
	W =  -167.362 deg,	P =    -0.003 deg,	R =  -159.248 deg
};
P[2655]{
   GP1:
	UF : 7, UT : 3,	CONFIG : 'F U T, 0, 0, 0',
	X =   -26.690  mm,	Y =   297.475  mm,	Z =     0.000  mm,
	W =  -167.362 deg,	P =    -0.003 deg,	R =  -159.248 deg
};
P[2656]{
   GP1:
	UF : 7, UT : 3,	CONFIG : 'F U T, 0, 0, 0',
	X =    26.690  mm,	Y =   297.475  mm,	Z =     0.000  mm,
	W =  -167.362 deg,	P =     0.001 deg,	R =  -170.599 deg
};
P[2657]{
   GP1:
	UF : 7, UT : 3,	CONFIG : 'F U T, 0, 0, 0',
	X =    26.690  mm,	Y =   297.475  mm,	Z =     0.000  mm,
	W =  -167.362 deg,	P =     0.001 deg,	R =  -170.599 deg
};
P[2658]{
   GP1:
	UF : 7, UT : 3,	CONFIG : 'F U T, 0, 0, 0',
	X =    26.690  mm,	Y =   297.475  mm,	Z =     0.000  mm,
	W =  -167.362 deg,	P =     0.001 deg,	R =  -170.599 deg
};
P[2659]{
   GP1:
	UF : 7, UT : 3,	CONFIG : 'F U T, 0, 0, 0',
	X =    26.690  mm,	Y =   297.475  mm,	Z =     0.000  mm,
	W =  -167.362 deg,	P =     0.001 deg,	R =  -170.599 deg
};
P[2660]{
   GP1:
	UF : 7, UT : 3,	CONFIG : 'F U T, 0, 0, 0',
	X =    48.017  mm,	Y =   294.772  mm,	Z =     0.001  mm,
	W =  -167.362 deg,	P =     0.000 deg,	R =  -174.233 deg
};
P[2661]{
   GP1:
	UF : 7, UT : 3,	CONFIG : 'F U T, 0, 0, 0',
	X =    67.443  mm,	Y =   290.948  mm,	Z =     0.001  mm,
	W =  -167.362 deg,	P =     0.000 deg,	R =  -177.997 deg
};
P[2662]{
   GP1:
	UF : 7, UT : 3,	CONFIG : 'F U T, 0, 0, 0',
	X =    86.518  mm,	Y =   285.853  mm,	Z =     0.000  mm,
	W =  -167.363 deg,	P =    -0.001 deg,	R =   178.233 deg
};
P[2663]{
   GP1:
	UF : 7, UT : 3,	CONFIG : 'F U T, 0, 0, 0',
	X =   105.027  mm,	Y =   279.584  mm,	Z =     0.000  mm,
	W =  -167.363 deg,	P =    -0.002 deg,	R =   174.416 deg
};
P[2664]{
   GP1:
	UF : 7, UT : 3,	CONFIG : 'F U T, 0, 0, 0',
	X =   105.027  mm,	Y =   279.584  mm,	Z =     0.000  mm,
	W =  -167.363 deg,	P =    -0.002 deg,	R =   174.416 deg
};
P[2665]{
   GP1:
	UF : 7, UT : 3,	CONFIG : 'F U T, 0, 0, 0',
	X =   105.027  mm,	Y =   279.584  mm,	Z =     0.000  mm,
	W =  -167.363 deg,	P =    -0.002 deg,	R =   174.416 deg
};
P[2666]{
   GP1:
	UF : 7, UT : 3,	CONFIG : 'F U T, 0, 0, 0',
	X =   105.027  mm,	Y =   279.584  mm,	Z =     0.000  mm,
	W =  -167.363 deg,	P =    -0.002 deg,	R =   174.416 deg
};
P[2667]{
   GP1:
	UF : 7, UT : 3,	CONFIG : 'F U T, 0, 0, 0',
	X =   153.101  mm,	Y =   256.429  mm,	Z =     0.000  mm,
	W =  -167.360 deg,	P =     0.002 deg,	R =   164.229 deg
};
P[2668]{
   GP1:
	UF : 7, UT : 3,	CONFIG : 'F U T, 0, 0, 0',
	X =   153.101  mm,	Y =   256.429  mm,	Z =     0.000  mm,
	W =  -167.360 deg,	P =     0.002 deg,	R =   164.229 deg
};
P[2669]{
   GP1:
	UF : 7, UT : 3,	CONFIG : 'F U T, 0, 0, 0',
	X =   153.101  mm,	Y =   256.429  mm,	Z =     0.000  mm,
	W =  -167.360 deg,	P =     0.002 deg,	R =   164.229 deg
};
P[2670]{
   GP1:
	UF : 7, UT : 3,	CONFIG : 'F U T, 0, 0, 0',
	X =   153.101  mm,	Y =   256.429  mm,	Z =     0.000  mm,
	W =  -167.360 deg,	P =     0.002 deg,	R =   164.229 deg
};
P[2671]{
   GP1:
	UF : 7, UT : 3,	CONFIG : 'F U T, 0, 0, 0',
	X =   170.045  mm,	Y =   245.526  mm,	Z =     0.001  mm,
	W =  -167.361 deg,	P =     0.001 deg,	R =   160.355 deg
};
P[2672]{
   GP1:
	UF : 7, UT : 3,	CONFIG : 'F U T, 0, 0, 0',
	X =   186.213  mm,	Y =   233.503  mm,	Z =     0.001  mm,
	W =  -167.362 deg,	P =     0.000 deg,	R =   156.480 deg
};
P[2673]{
   GP1:
	UF : 7, UT : 3,	CONFIG : 'F U T, 0, 0, 0',
	X =   201.532  mm,	Y =   220.414  mm,	Z =     0.001  mm,
	W =  -167.362 deg,	P =    -0.002 deg,	R =   152.606 deg
};
P[2674]{
   GP1:
	UF : 7, UT : 3,	CONFIG : 'F U T, 0, 0, 0',
	X =   215.932  mm,	Y =   206.321  mm,	Z =     0.000  mm,
	W =  -167.362 deg,	P =    -0.003 deg,	R =   148.732 deg
};
P[2675]{
   GP1:
	UF : 7, UT : 3,	CONFIG : 'F U T, 0, 0, 0',
	X =   215.932  mm,	Y =   206.321  mm,	Z =     0.000  mm,
	W =  -167.362 deg,	P =    -0.003 deg,	R =   148.732 deg
};
P[2676]{
   GP1:
	UF : 7, UT : 3,	CONFIG : 'F U T, 0, 0, 0',
	X =   215.932  mm,	Y =   206.321  mm,	Z =     0.000  mm,
	W =  -167.362 deg,	P =    -0.003 deg,	R =   148.732 deg
};
P[2677]{
   GP1:
	UF : 7, UT : 3,	CONFIG : 'F U T, 0, 0, 0',
	X =   215.932  mm,	Y =   206.321  mm,	Z =     0.000  mm,
	W =  -167.362 deg,	P =    -0.003 deg,	R =   148.732 deg
};
P[2678]{
   GP1:
	UF : 7, UT : 3,	CONFIG : 'F U T, 0, 0, 0',
	X =   249.198  mm,	Y =   164.607  mm,	Z =     0.000  mm,
	W =  -167.360 deg,	P =     0.003 deg,	R =   138.993 deg
};
P[2679]{
   GP1:
	UF : 7, UT : 3,	CONFIG : 'F U T, 0, 0, 0',
	X =   249.198  mm,	Y =   164.607  mm,	Z =     0.000  mm,
	W =  -167.360 deg,	P =     0.003 deg,	R =   138.993 deg
};
P[2680]{
   GP1:
	UF : 7, UT : 3,	CONFIG : 'F U T, 0, 0, 0',
	X =   249.198  mm,	Y =   164.607  mm,	Z =     0.000  mm,
	W =  -167.360 deg,	P =     0.003 deg,	R =   138.993 deg
};
P[2681]{
   GP1:
	UF : 7, UT : 3,	CONFIG : 'F U T, 0, 0, 0',
	X =   249.198  mm,	Y =   164.607  mm,	Z =     0.000  mm,
	W =  -167.360 deg,	P =     0.003 deg,	R =   138.993 deg
};
P[2682]{
   GP1:
	UF : 7, UT : 3,	CONFIG : 'F U T, 0, 0, 0',
	X =   259.274  mm,	Y =   148.234  mm,	Z =     0.001  mm,
	W =  -167.361 deg,	P =     0.001 deg,	R =   134.846 deg
};
P[2683]{
   GP1:
	UF : 7, UT : 3,	CONFIG : 'F U T, 0, 0, 0',
	X =   268.685  mm,	Y =   130.404  mm,	Z =     0.002  mm,
	W =  -167.361 deg,	P =     0.000 deg,	R =   130.951 deg
};
P[2684]{
   GP1:
	UF : 7, UT : 3,	CONFIG : 'F U T, 0, 0, 0',
	X =   276.904  mm,	Y =   111.895  mm,	Z =     0.001  mm,
	W =  -167.362 deg,	P =    -0.001 deg,	R =   127.076 deg
};
P[2685]{
   GP1:
	UF : 7, UT : 3,	CONFIG : 'F U T, 0, 0, 0',
	X =   284.072  mm,	Y =    92.207  mm,	Z =     0.000  mm,
	W =  -167.362 deg,	P =    -0.003 deg,	R =   123.285 deg
};
P[2686]{
   GP1:
	UF : 7, UT : 3,	CONFIG : 'F U T, 0, 0, 0',
	X =   284.072  mm,	Y =    92.207  mm,	Z =     0.000  mm,
	W =  -167.362 deg,	P =    -0.003 deg,	R =   123.285 deg
};
P[2687]{
   GP1:
	UF : 7, UT : 3,	CONFIG : 'F U T, 0, 0, 0',
	X =   284.072  mm,	Y =    92.207  mm,	Z =     0.000  mm,
	W =  -167.362 deg,	P =    -0.003 deg,	R =   123.285 deg
};
P[2688]{
   GP1:
	UF : 7, UT : 3,	CONFIG : 'F U T, 0, 0, 0',
	X =   284.072  mm,	Y =    92.207  mm,	Z =     0.000  mm,
	W =  -167.362 deg,	P =    -0.003 deg,	R =   123.285 deg
};
P[2689]{
   GP1:
	UF : 7, UT : 3,	CONFIG : 'F U T, 0, 0, 0',
	X =   295.952  mm,	Y =    40.176  mm,	Z =     0.000  mm,
	W =  -167.362 deg,	P =     0.001 deg,	R =   112.465 deg
};
P[2690]{
   GP1:
	UF : 7, UT : 3,	CONFIG : 'F U T, 0, 0, 0',
	X =   295.952  mm,	Y =    40.176  mm,	Z =     0.000  mm,
	W =  -167.362 deg,	P =     0.001 deg,	R =   112.465 deg
};
P[2691]{
   GP1:
	UF : 7, UT : 3,	CONFIG : 'F U T, 0, 0, 0',
	X =   295.952  mm,	Y =    40.176  mm,	Z =     0.000  mm,
	W =  -167.362 deg,	P =     0.001 deg,	R =   112.465 deg
};
P[2692]{
   GP1:
	UF : 7, UT : 3,	CONFIG : 'F U T, 0, 0, 0',
	X =   295.952  mm,	Y =    40.176  mm,	Z =     0.000  mm,
	W =  -167.362 deg,	P =     0.001 deg,	R =   112.465 deg
};
P[2693]{
   GP1:
	UF : 7, UT : 3,	CONFIG : 'F U T, 0, 0, 0',
	X =   297.936  mm,	Y =    20.868  mm,	Z =     0.000  mm,
	W =  -167.363 deg,	P =     0.000 deg,	R =   109.073 deg
};
P[2694]{
   GP1:
	UF : 7, UT : 3,	CONFIG : 'F U T, 0, 0, 0',
	X =   298.673  mm,	Y =     0.000  mm,	Z =     0.000  mm,
	W =  -167.364 deg,	P =    -0.001 deg,	R =   105.700 deg
};
P[2695]{
   GP1:
	UF : 7, UT : 3,	CONFIG : 'F U T, 0, 0, 0',
	X =   298.673  mm,	Y =     0.000  mm,	Z =     0.000  mm,
	W =  -167.364 deg,	P =    -0.001 deg,	R =   105.700 deg
};
P[2696]{
   GP1:
	UF : 7, UT : 3,	CONFIG : 'F U T, 0, 0, 0',
	X =   298.673  mm,	Y =     0.000  mm,	Z =     0.000  mm,
	W =  -167.364 deg,	P =    -0.001 deg,	R =   105.700 deg
};
P[2697]{
   GP1:
	UF : 7, UT : 3,	CONFIG : 'F U T, 0, 0, 0',
	X =   298.673  mm,	Y =     0.000  mm,	Z =     0.000  mm,
	W =  -167.364 deg,	P =    -0.001 deg,	R =   105.700 deg
};
P[2698]{
   GP1:
	UF : 7, UT : 3,	CONFIG : 'F U T, 0, 0, 0',
	X =   295.539  mm,	Y =     0.000  mm,	Z =     0.000  mm,
	W =  -167.364 deg,	P =    -0.001 deg,	R =   105.697 deg
};
P[2699]{
   GP1:
	UF : 7, UT : 3,	CONFIG : 'F U T, 0, 0, 0',
	X =   295.539  mm,	Y =     0.000  mm,	Z =     0.000  mm,
	W =  -167.364 deg,	P =    -0.001 deg,	R =   105.697 deg
};
P[2700]{
   GP1:
	UF : 7, UT : 3,	CONFIG : 'F U T, 0, 0, 0',
	X =   295.539  mm,	Y =     0.000  mm,	Z =     0.000  mm,
	W =  -167.364 deg,	P =    -0.001 deg,	R =   105.697 deg
};
P[2701]{
   GP1:
	UF : 7, UT : 3,	CONFIG : 'F U T, 0, 0, 0',
	X =   295.539  mm,	Y =     0.000  mm,	Z =     0.000  mm,
	W =  -167.364 deg,	P =    -0.001 deg,	R =   105.697 deg
};
P[2702]{
   GP1:
	UF : 7, UT : 3,	CONFIG : 'F U T, 0, 0, 0',
	X =   294.616  mm,	Y =    23.147  mm,	Z =     0.000  mm,
	W =  -167.363 deg,	P =     0.000 deg,	R =   109.538 deg
};
P[2703]{
   GP1:
	UF : 7, UT : 3,	CONFIG : 'F U T, 0, 0, 0',
	X =   292.447  mm,	Y =    42.514  mm,	Z =     0.000  mm,
	W =  -167.362 deg,	P =     0.001 deg,	R =   113.811 deg
};
P[2704]{
   GP1:
	UF : 7, UT : 3,	CONFIG : 'F U T, 0, 0, 0',
	X =   292.447  mm,	Y =    42.514  mm,	Z =     0.000  mm,
	W =  -167.362 deg,	P =     0.001 deg,	R =   113.811 deg
};
P[2705]{
   GP1:
	UF : 7, UT : 3,	CONFIG : 'F U T, 0, 0, 0',
	X =   292.447  mm,	Y =    42.514  mm,	Z =     0.000  mm,
	W =  -167.362 deg,	P =     0.001 deg,	R =   113.811 deg
};
P[2706]{
   GP1:
	UF : 7, UT : 3,	CONFIG : 'F U T, 0, 0, 0',
	X =   292.447  mm,	Y =    42.514  mm,	Z =     0.000  mm,
	W =  -167.362 deg,	P =     0.001 deg,	R =   113.811 deg
};
P[2707]{
   GP1:
	UF : 7, UT : 3,	CONFIG : 'F U T, 0, 0, 0',
	X =   281.935  mm,	Y =    88.590  mm,	Z =     0.000  mm,
	W =  -167.362 deg,	P =    -0.002 deg,	R =   122.465 deg
};
P[2708]{
   GP1:
	UF : 7, UT : 3,	CONFIG : 'F U T, 0, 0, 0',
	X =   281.935  mm,	Y =    88.590  mm,	Z =     0.000  mm,
	W =  -167.362 deg,	P =    -0.002 deg,	R =   122.465 deg
};
P[2709]{
   GP1:
	UF : 7, UT : 3,	CONFIG : 'F U T, 0, 0, 0',
	X =   281.935  mm,	Y =    88.590  mm,	Z =     0.000  mm,
	W =  -167.362 deg,	P =    -0.002 deg,	R =   122.465 deg
};
P[2710]{
   GP1:
	UF : 7, UT : 3,	CONFIG : 'F U T, 0, 0, 0',
	X =   281.935  mm,	Y =    88.590  mm,	Z =     0.000  mm,
	W =  -167.362 deg,	P =    -0.002 deg,	R =   122.465 deg
};
P[2711]{
   GP1:
	UF : 7, UT : 3,	CONFIG : 'F U T, 0, 0, 0',
	X =   274.907  mm,	Y =   108.481  mm,	Z =     0.001  mm,
	W =  -167.362 deg,	P =    -0.001 deg,	R =   126.587 deg
};
P[2712]{
   GP1:
	UF : 7, UT : 3,	CONFIG : 'F U T, 0, 0, 0',
	X =   266.447  mm,	Y =   127.830  mm,	Z =     0.002  mm,
	W =  -167.361 deg,	P =     0.000 deg,	R =   130.703 deg
};
P[2713]{
   GP1:
	UF : 7, UT : 3,	CONFIG : 'F U T, 0, 0, 0',
	X =   256.518  mm,	Y =   146.734  mm,	Z =     0.001  mm,
	W =  -167.360 deg,	P =     0.001 deg,	R =   134.776 deg
};
P[2714]{
   GP1:
	UF : 7, UT : 3,	CONFIG : 'F U T, 0, 0, 0',
	X =   245.049  mm,	Y =   165.190  mm,	Z =     0.000  mm,
	W =  -167.360 deg,	P =     0.002 deg,	R =   138.811 deg
};
P[2715]{
   GP1:
	UF : 7, UT : 3,	CONFIG : 'F U T, 0, 0, 0',
	X =   245.049  mm,	Y =   165.190  mm,	Z =     0.000  mm,
	W =  -167.360 deg,	P =     0.002 deg,	R =   138.811 deg
};
P[2716]{
   GP1:
	UF : 7, UT : 3,	CONFIG : 'F U T, 0, 0, 0',
